LIN {X 0,Y 249.727,Z 1176.579,A -85,B 0,C 180,E1 12706.065,E2 12706.065} C_VEL
LIN {X 0,Y 248.616,Z 1179.166,A -85,B 0,C 180,E1 12701.365,E2 12701.365} C_VEL
LIN {X 0,Y 248.168,Z 1180.788,A -85,B 0,C 180,E1 12696.942,E2 12696.942} C_VEL
LIN {X 0,Y 248.027,Z 1181.611,A -85,B 0,C 180,E1 12692.773,E2 12692.773} C_VEL
LIN {X 0,Y 248.02,Z 1181.751,A -85,B 0,C 180,E1 12688.614,E2 12688.614} C_VEL
LIN {X 0,Y 248.114,Z 1181.08,A -85,B 0,C 180,E1 12683.986,E2 12683.986} C_VEL
LIN {X 0,Y 248.534,Z 1179.438,A -85,B 0,C 180,E1 12679.101,E2 12679.101} C_VEL
LIN {X 0,Y 249.624,Z 1176.826,A -85,B 0,C 180,E1 12674.195,E2 12674.195} C_VEL
LIN {X 0,Y 251.654,Z 1173.217,A -85,B 0,C 180,E1 12669.292,E2 12669.292} C_VEL
LIN {X 0,Y 254.855,Z 1168.577,A -85,B 0,C 180,E1 12664.434,E2 12664.434} C_VEL
LIN {X 0,Y 259.34,Z 1162.869,A -85,B 0,C 180,E1 12659.665,E2 12659.665} C_VEL
LIN {X 0,Y 266.478,Z 1154.638,A -85,B 0,C 180,E1 12654.144,E2 12654.144} C_VEL
LIN {X 0,Y 275.857,Z 1144.197,A -85,B 0,C 180,E1 12648.726,E2 12648.726} C_VEL
LIN {X 0,Y 284.944,Z 1134.318,A -85,B 0,C 180,E1 12644.573,E2 12644.573} C_VEL
LIN {X 0,Y 294.763,Z 1123.639,A -85,B 0,C 180,E1 12640.849,E2 12640.849} C_VEL
LIN {X 0,Y 307.374,Z 1109.73,A -85,B 0,C 180,E1 12636.85,E2 12636.85} C_VEL
LIN {X 0,Y 320.654,Z 1094.237,A -85,B 0,C 180,E1 12633.286,E2 12633.286} C_VEL
LIN {X 0,Y 332.217,Z 1080.145,A -85,B 0,C 180,E1 12630.598,E2 12630.598} C_VEL
LIN {X 0,Y 343.091,Z 1066.216,A -85,B 0,C 180,E1 12628.345,E2 12628.345} C_VEL
LIN {X 0,Y 354.794,Z 1050.336,A -85,B 0,C 180,E1 12626.159,E2 12626.159} C_VEL
LIN {X 0,Y 368.74,Z 1030.057,A -85,B 0,C 180,E1 12623.831,E2 12623.831} C_VEL
LIN {X 0,Y 381.488,Z 1009.491,A -85,B 0,C 180,E1 12621.904,E2 12621.904} C_VEL
LIN {X 0,Y 391.938,Z 991.177,A -85,B 0,C 180,E1 12620.457,E2 12620.457} C_VEL
LIN {X 0,Y 401.368,Z 973.16,A -85,B 0,C 180,E1 12619.242,E2 12619.242} C_VEL
LIN {X 0,Y 411.167,Z 952.497,A -85,B 0,C 180,E1 12618.045,E2 12618.045} C_VEL
LIN {X 0,Y 422.058,Z 926.302,A -85,B 0,C 180,E1 12616.8,E2 12616.8} C_VEL
LIN {X 0,Y 429.551,Z 905.47,A -85,B 0,C 180,E1 12615.986,E2 12615.986} C_VEL
LIN {X 0,Y 435.925,Z 885.156,A -85,B 0,C 180,E1 12615.318,E2 12615.318} C_VEL
LIN {X 0,Y 441.618,Z 863.935,A -85,B 0,C 180,E1 12614.735,E2 12614.735} C_VEL
LIN {X 0,Y 445.99,Z 844.495,A -85,B 0,C 180,E1 12614.298,E2 12614.298} C_VEL
LIN {X 0,Y 447.312,Z 837.117,A -85,B 0,C 180,E1 12614.033,E2 12614.033} C_VEL
LIN {X 0,Y 449.125,Z 817.839,A -85,B 0,C 180,E1 12612.916,E2 12612.916} C_VEL
LIN {X 0,Y 449.804,Z 811.396,A -85,B 0,C 180,E1 12612.724,E2 12612.724} C_VEL
LIN {X 0,Y 456.299,Z 750.449,A -85,B 0,C 180,E1 12611.84,E2 12611.84} C_VEL
LIN {X 0,Y 471.03,Z 607.918,A -85,B 0,C 180,E1 12609.811,E2 12609.811} C_VEL
LIN {X 0,Y 468.952,Z 603.858,A -85,B 0,C 180,E1 12607.72,E2 12607.72} C_VEL
LIN {X 0,Y 467.352,Z 600.49,A -85,B 0,C 180,E1 12605.525,E2 12605.525} C_VEL
LIN {X 0,Y 465.914,Z 596.286,A -85,B 0,C 180,E1 12601.107,E2 12601.107} C_VEL
LIN {X 0,Y 465.917,Z 596.314,A -85,B 0,C 180,E1 12599.262,E2 12599.262} C_VEL
LIN {X 0,Y 467.226,Z 600.314,A -85,B 0,C 180,E1 12595.089,E2 12595.089} C_VEL
LIN {X 0,Y 467.857,Z 601.547,A -85,B 0,C 180,E1 12594.112,E2 12594.112} C_VEL
LIN {X 0,Y 470.021,Z 605.91,A -85,B 0,C 180,E1 12591.559,E2 12591.559} C_VEL
LIN {X 0,Y 471.151,Z 608.251,A -85,B 0,C 180,E1 12590.489,E2 12590.489} C_VEL
LIN {X 0,Y 449.874,Z 813.61,A -85,B 0,C 180,E1 12587.551,E2 12587.551} C_VEL
LIN {X 0,Y 446.454,Z 836.613,A -85,B 0,C 180,E1 12587.182,E2 12587.182} C_VEL
LIN {X 0,Y 440.618,Z 864.958,A -85,B 0,C 180,E1 12586.666,E2 12586.666} C_VEL
LIN {X 0,Y 434.14,Z 889.147,A -85,B 0,C 180,E1 12586.106,E2 12586.106} C_VEL
LIN {X 0,Y 427.55,Z 910.072,A -85,B 0,C 180,E1 12585.504,E2 12585.504} C_VEL
LIN {X 0,Y 420.15,Z 930.562,A -85,B 0,C 180,E1 12584.794,E2 12584.794} C_VEL
LIN {X 0,Y 411.591,Z 951.546,A -85,B 0,C 180,E1 12583.922,E2 12583.922} C_VEL
LIN {X 0,Y 399.271,Z 978.022,A -85,B 0,C 180,E1 12582.573,E2 12582.573} C_VEL
LIN {X 0,Y 388.486,Z 998.548,A -85,B 0,C 180,E1 12581.286,E2 12581.286} C_VEL
LIN {X 0,Y 378.298,Z 1016.269,A -85,B 0,C 180,E1 12579.984,E2 12579.984} C_VEL
LIN {X 0,Y 367.137,Z 1034.234,A -85,B 0,C 180,E1 12578.428,E2 12578.428} C_VEL
LIN {X 0,Y 353.455,Z 1054.661,A -85,B 0,C 180,E1 12576.315,E2 12576.315} C_VEL
LIN {X 0,Y 338.832,Z 1074.514,A -85,B 0,C 180,E1 12573.776,E2 12573.776} C_VEL
LIN {X 0,Y 326.822,Z 1089.878,A -85,B 0,C 180,E1 12571.405,E2 12571.405} C_VEL
LIN {X 0,Y 315.399,Z 1103.791,A -85,B 0,C 180,E1 12568.863,E2 12568.863} C_VEL
LIN {X 0,Y 303.391,Z 1117.825,A -85,B 0,C 180,E1 12565.812,E2 12565.812} C_VEL
LIN {X 0,Y 288.384,Z 1134.661,A -85,B 0,C 180,E1 12561.269,E2 12561.269} C_VEL
LIN {X 0,Y 277.619,Z 1146.477,A -85,B 0,C 180,E1 12557.283,E2 12557.283} C_VEL
LIN {X 0,Y 268.578,Z 1156.436,A -85,B 0,C 180,E1 12553.235,E2 12553.235} C_VEL
LIN {X 0,Y 260.061,Z 1166.03,A -85,B 0,C 180,E1 12548.524,E2 12548.524} C_VEL
LIN {X 0,Y 251.434,Z 1176.35,A -85,B 0,C 180,E1 12542.107,E2 12542.107} C_VEL
LIN {X 0,Y 246.423,Z 1183.046,A -85,B 0,C 180,E1 12536.768,E2 12536.768} C_VEL
LIN {X 0,Y 243.201,Z 1188.116,A -85,B 0,C 180,E1 12531.716,E2 12531.716} C_VEL
LIN {X 0,Y 241.293,Z 1191.973,A -85,B 0,C 180,E1 12526.815,E2 12526.815} C_VEL
LIN {X 0,Y 240.319,Z 1194.802,A -85,B 0,C 180,E1 12522.007,E2 12522.007} C_VEL
LIN {X 0,Y 240.037,Z 1196.639,A -85,B 0,C 180,E1 12517.419,E2 12517.419} C_VEL
LIN {X 0,Y 240.009,Z 1197.592,A -85,B 0,C 180,E1 12513.104,E2 12513.104} C_VEL
LIN {X 0,Y 240.02,Z 1197.782,A -85,B 0,C 180,E1 12508.807,E2 12508.807} C_VEL
LIN {X 0,Y 240.006,Z 1197.061,A -85,B 0,C 180,E1 12504.022,E2 12504.022} C_VEL
LIN {X 0,Y 240.223,Z 1195.267,A -85,B 0,C 180,E1 12498.962,E2 12498.962} C_VEL
LIN {X 0,Y 241.106,Z 1192.425,A -85,B 0,C 180,E1 12493.868,E2 12493.868} C_VEL
LIN {X 0,Y 242.957,Z 1188.524,A -85,B 0,C 180,E1 12488.768,E2 12488.768} C_VEL
LIN {X 0,Y 246.061,Z 1183.545,A -85,B 0,C 180,E1 12483.71,E2 12483.71} C_VEL
LIN {X 0,Y 250.51,Z 1177.46,A -85,B 0,C 180,E1 12478.744,E2 12478.744} C_VEL
LIN {X 0,Y 257.044,Z 1169.504,A -85,B 0,C 180,E1 12473.477,E2 12473.477} C_VEL
LIN {X 0,Y 267.323,Z 1157.79,A -85,B 0,C 180,E1 12467.392,E2 12467.392} C_VEL
LIN {X 0,Y 276.776,Z 1147.339,A -85,B 0,C 180,E1 12463.062,E2 12463.062} C_VEL
LIN {X 0,Y 286.761,Z 1136.342,A -85,B 0,C 180,E1 12459.281,E2 12459.281} C_VEL
LIN {X 0,Y 299.166,Z 1122.555,A -85,B 0,C 180,E1 12455.365,E2 12455.365} C_VEL
LIN {X 0,Y 313.835,Z 1105.53,A -85,B 0,C 180,E1 12451.501,E2 12451.501} C_VEL
LIN {X 0,Y 326.118,Z 1090.599,A -85,B 0,C 180,E1 12448.735,E2 12448.735} C_VEL
LIN {X 0,Y 338.094,Z 1075.298,A -85,B 0,C 180,E1 12446.354,E2 12446.354} C_VEL
LIN {X 0,Y 352.128,Z 1056.313,A -85,B 0,C 180,E1 12443.892,E2 12443.892} C_VEL
LIN {X 0,Y 366.36,Z 1035.204,A -85,B 0,C 180,E1 12441.677,E2 12441.677} C_VEL
LIN {X 0,Y 377.88,Z 1016.689,A -85,B 0,C 180,E1 12440.063,E2 12440.063} C_VEL
LIN {X 0,Y 388.469,Z 998.262,A -85,B 0,C 180,E1 12438.707,E2 12438.707} C_VEL
LIN {X 0,Y 399.677,Z 976.889,A -85,B 0,C 180,E1 12437.373,E2 12437.373} C_VEL
LIN {X 0,Y 411.443,Z 951.467,A -85,B 0,C 180,E1 12436.084,E2 12436.084} C_VEL
LIN {X 0,Y 420.134,Z 930.114,A -85,B 0,C 180,E1 12435.197,E2 12435.197} C_VEL
LIN {X 0,Y 427.534,Z 909.552,A -85,B 0,C 180,E1 12434.487,E2 12434.487} C_VEL
LIN {X 0,Y 434.347,Z 887.8,A -85,B 0,C 180,E1 12433.867,E2 12433.867} C_VEL
LIN {X 0,Y 441.555,Z 860.083,A -85,B 0,C 180,E1 12433.243,E2 12433.243} C_VEL
LIN {X 0,Y 446.555,Z 834.801,A -85,B 0,C 180,E1 12432.794,E2 12432.794} C_VEL
LIN {X 0,Y 449.81,Z 812.463,A -85,B 0,C 180,E1 12432.437,E2 12432.437} C_VEL
LIN {X 0,Y 470.962,Z 607.908,A -85,B 0,C 180,E1 12429.509,E2 12429.509} C_VEL
LIN {X 0,Y 468.889,Z 603.932,A -85,B 0,C 180,E1 12427.474,E2 12427.474} C_VEL
LIN {X 0,Y 467.155,Z 600.324,A -85,B 0,C 180,E1 12425.158,E2 12425.158} C_VEL
LIN {X 0,Y 465.714,Z 596.603,A -85,B 0,C 180,E1 12421.353,E2 12421.353} C_VEL
LIN {X 0,Y 465.647,Z 596.093,A -85,B 0,C 180,E1 12420.615,E2 12420.615} C_VEL
LIN {X 0,Y 465.682,Z 596.236,A -85,B 0,C 180,E1 12418.524,E2 12418.524} C_VEL
LIN {X 0,Y 467.54,Z 601.157,A -85,B 0,C 180,E1 12413.738,E2 12413.738} C_VEL
LIN {X 0,Y 469.614,Z 605.388,A -85,B 0,C 180,E1 12411.243,E2 12411.243} C_VEL
LIN {X 0,Y 470.81,Z 607.98,A -85,B 0,C 180,E1 12410.086,E2 12410.086} C_VEL
LIN {X 0,Y 449.965,Z 808.417,A -85,B 0,C 180,E1 12407.225,E2 12407.225} C_VEL
LIN {X 0,Y 446.124,Z 833.492,A -85,B 0,C 180,E1 12406.821,E2 12406.821} C_VEL
LIN {X 0,Y 440.07,Z 861.713,A -85,B 0,C 180,E1 12406.239,E2 12406.239} C_VEL
LIN {X 0,Y 434.212,Z 883.569,A -85,B 0,C 180,E1 12405.663,E2 12405.663} C_VEL
LIN {X 0,Y 427.959,Z 903.481,A -85,B 0,C 180,E1 12405.033,E2 12405.033} C_VEL
LIN {X 0,Y 420.689,Z 923.691,A -85,B 0,C 180,E1 12404.273,E2 12404.273} C_VEL
LIN {X 0,Y 411.386,Z 946.458,A -85,B 0,C 180,E1 12403.256,E2 12403.256} C_VEL
LIN {X 0,Y 399.73,Z 971.175,A -85,B 0,C 180,E1 12401.898,E2 12401.898} C_VEL
LIN {X 0,Y 389.529,Z 990.45,A -85,B 0,C 180,E1 12400.637,E2 12400.637} C_VEL
LIN {X 0,Y 379.06,Z 1008.555,A -85,B 0,C 180,E1 12399.24,E2 12399.24} C_VEL
LIN {X 0,Y 367.699,Z 1026.642,A -85,B 0,C 180,E1 12397.598,E2 12397.598} C_VEL
LIN {X 0,Y 352.89,Z 1048.188,A -85,B 0,C 180,E1 12395.242,E2 12395.242} C_VEL
LIN {X 0,Y 340.117,Z 1065.189,A -85,B 0,C 180,E1 12392.966,E2 12392.966} C_VEL
LIN {X 0,Y 328.91,Z 1079.228,A -85,B 0,C 180,E1 12390.745,E2 12390.745} C_VEL
LIN {X 0,Y 317.549,Z 1092.731,A -85,B 0,C 180,E1 12388.227,E2 12388.227} C_VEL
LIN {X 0,Y 305.594,Z 1106.31,A -85,B 0,C 180,E1 12385.208,E2 12385.208} C_VEL
LIN {X 0,Y 291.164,Z 1121.982,A -85,B 0,C 180,E1 12380.903,E2 12380.903} C_VEL
LIN {X 0,Y 280.268,Z 1133.369,A -85,B 0,C 180,E1 12376.999,E2 12376.999} C_VEL
LIN {X 0,Y 271.036,Z 1142.926,A -85,B 0,C 180,E1 12373.037,E2 12373.037} C_VEL
LIN {X 0,Y 262.669,Z 1151.691,A -85,B 0,C 180,E1 12368.629,E2 12368.629} C_VEL
LIN {X 0,Y 254.223,Z 1160.944,A -85,B 0,C 180,E1 12362.871,E2 12362.871} C_VEL
LIN {X 0,Y 247.901,Z 1168.239,A -85,B 0,C 180,E1 12356.855,E2 12356.855} C_VEL
LIN {X 0,Y 244.17,Z 1173.191,A -85,B 0,C 180,E1 12351.626,E2 12351.626} C_VEL
LIN {X 0,Y 241.887,Z 1176.865,A -85,B 0,C 180,E1 12346.572,E2 12346.572} C_VEL
LIN {X 0,Y 240.683,Z 1179.432,A -85,B 0,C 180,E1 12341.745,E2 12341.745} C_VEL
LIN {X 0,Y 240.186,Z 1181.052,A -85,B 0,C 180,E1 12337.174,E2 12337.174} C_VEL
LIN {X 0,Y 240.033,Z 1181.874,A -85,B 0,C 180,E1 12332.865,E2 12332.865} C_VEL
LIN {X 0,Y 240.025,Z 1182.013,A -85,B 0,C 180,E1 12328.568,E2 12328.568} C_VEL
LIN {X 0,Y 240.129,Z 1181.343,A -85,B 0,C 180,E1 12323.785,E2 12323.785} C_VEL
LIN {X 0,Y 240.592,Z 1179.703,A -85,B 0,C 180,E1 12318.736,E2 12318.736} C_VEL
LIN {X 0,Y 241.801,Z 1177.057,A -85,B 0,C 180,E1 12313.611,E2 12313.611} C_VEL
LIN {X 0,Y 243.989,Z 1173.486,A -85,B 0,C 180,E1 12308.61,E2 12308.61} C_VEL
LIN {X 0,Y 247.426,Z 1168.847,A -85,B 0,C 180,E1 12303.608,E2 12303.608} C_VEL
LIN {X 0,Y 252.207,Z 1163.141,A -85,B 0,C 180,E1 12298.712,E2 12298.712} C_VEL
LIN {X 0,Y 259.734,Z 1154.949,A -85,B 0,C 180,E1 12293.092,E2 12293.092} C_VEL
LIN {X 0,Y 269.634,Z 1144.47,A -85,B 0,C 180,E1 12287.554,E2 12287.554} C_VEL
LIN {X 0,Y 279.146,Z 1134.596,A -85,B 0,C 180,E1 12283.355,E2 12283.355} C_VEL
LIN {X 0,Y 289.38,Z 1123.911,A -85,B 0,C 180,E1 12279.601,E2 12279.601} C_VEL
LIN {X 0,Y 302.487,Z 1109.963,A -85,B 0,C 180,E1 12275.576,E2 12275.576} C_VEL
LIN {X 0,Y 316.108,Z 1094.573,A -85,B 0,C 180,E1 12272.039,E2 12272.039} C_VEL
LIN {X 0,Y 328.073,Z 1080.415,A -85,B 0,C 180,E1 12269.351,E2 12269.351} C_VEL
LIN {X 0,Y 339.246,Z 1066.484,A -85,B 0,C 180,E1 12267.117,E2 12267.117} C_VEL
LIN {X 0,Y 350.868,Z 1051.103,A -85,B 0,C 180,E1 12265.016,E2 12265.016} C_VEL
LIN {X 0,Y 365.112,Z 1030.929,A -85,B 0,C 180,E1 12262.715,E2 12262.715} C_VEL
LIN {X 0,Y 378.514,Z 1009.755,A -85,B 0,C 180,E1 12260.756,E2 12260.756} C_VEL
LIN {X 0,Y 388.941,Z 991.838,A -85,B 0,C 180,E1 12259.361,E2 12259.361} C_VEL
LIN {X 0,Y 398.351,Z 974.227,A -85,B 0,C 180,E1 12258.19,E2 12258.19} C_VEL
LIN {X 0,Y 407.47,Z 955.44,A -85,B 0,C 180,E1 12257.107,E2 12257.107} C_VEL
LIN {X 0,Y 418.014,Z 931.249,A -85,B 0,C 180,E1 12255.94,E2 12255.94} C_VEL
LIN {X 0,Y 426.974,Z 907.004,A -85,B 0,C 180,E1 12254.992,E2 12254.992} C_VEL
LIN {X 0,Y 433.654,Z 886.148,A -85,B 0,C 180,E1 12254.315,E2 12254.315} C_VEL
LIN {X 0,Y 439.482,Z 864.836,A -85,B 0,C 180,E1 12253.739,E2 12253.739} C_VEL
LIN {X 0,Y 444.549,Z 842.515,A -85,B 0,C 180,E1 12253.252,E2 12253.252} C_VEL
LIN {X 0,Y 449.48,Z 814.028,A -85,B 0,C 180,E1 12252.763,E2 12252.763} C_VEL
LIN {X 0,Y 449.804,Z 811.396,A -85,B 0,C 180,E1 12252.724,E2 12252.724} C_VEL
LIN {X 0,Y 450.526,Z 803.885,A -85,B 0,C 180,E1 12252.49,E2 12252.49} C_VEL
LIN {X 0,Y 451.401,Z 784.372,A -85,B 0,C 180,E1 12251.427,E2 12251.427} C_VEL
LIN {X 0,Y 451.905,Z 777.899,A -85,B 0,C 180,E1 12251.237,E2 12251.237} C_VEL
LIN {X 0,Y 469.061,Z 614.281,A -85,B 0,C 180,E1 12248.921,E2 12248.921} C_VEL
LIN {X 0,Y 467.756,Z 611.57,A -85,B 0,C 180,E1 12247.492,E2 12247.492} C_VEL
LIN {X 0,Y 466.218,Z 608.279,A -85,B 0,C 180,E1 12245.291,E2 12245.291} C_VEL
LIN {X 0,Y 464.923,Z 604.057,A -85,B 0,C 180,E1 12240.739,E2 12240.739} C_VEL
LIN {X 0,Y 464.933,Z 604.329,A -85,B 0,C 180,E1 12239.261,E2 12239.261} C_VEL
LIN {X 0,Y 466.251,Z 608.287,A -85,B 0,C 180,E1 12235.079,E2 12235.079} C_VEL
LIN {X 0,Y 466.989,Z 609.985,A -85,B 0,C 180,E1 12233.916,E2 12233.916} C_VEL
LIN {X 0,Y 468.79,Z 613.597,A -85,B 0,C 180,E1 12231.784,E2 12231.784} C_VEL
LIN {X 0,Y 469.179,Z 614.647,A -85,B 0,C 180,E1 12231.366,E2 12231.366} C_VEL
LIN {X 0,Y 448.075,Z 814.43,A -85,B 0,C 180,E1 12228.541,E2 12228.541} C_VEL
LIN {X 0,Y 444.253,Z 839.22,A -85,B 0,C 180,E1 12228.147,E2 12228.147} C_VEL
LIN {X 0,Y 437.953,Z 868.083,A -85,B 0,C 180,E1 12227.62,E2 12227.62} C_VEL
LIN {X 0,Y 432.048,Z 889.633,A -85,B 0,C 180,E1 12227.127,E2 12227.127} C_VEL
LIN {X 0,Y 425.417,Z 910.328,A -85,B 0,C 180,E1 12226.545,E2 12226.545} C_VEL
LIN {X 0,Y 417.653,Z 931.439,A -85,B 0,C 180,E1 12225.827,E2 12225.827} C_VEL
LIN {X 0,Y 407.204,Z 956.413,A -85,B 0,C 180,E1 12224.792,E2 12224.792} C_VEL
LIN {X 0,Y 396.041,Z 979.393,A -85,B 0,C 180,E1 12223.609,E2 12223.609} C_VEL
LIN {X 0,Y 385.924,Z 998.282,A -85,B 0,C 180,E1 12222.443,E2 12222.443} C_VEL
LIN {X 0,Y 375.549,Z 1016.001,A -85,B 0,C 180,E1 12221.169,E2 12221.169} C_VEL
LIN {X 0,Y 364.195,Z 1033.929,A -85,B 0,C 180,E1 12219.644,E2 12219.644} C_VEL
LIN {X 0,Y 350.017,Z 1054.65,A -85,B 0,C 180,E1 12217.534,E2 12217.534} C_VEL
LIN {X 0,Y 335.031,Z 1074.483,A -85,B 0,C 180,E1 12215.024,E2 12215.024} C_VEL
LIN {X 0,Y 322.893,Z 1089.606,A -85,B 0,C 180,E1 12212.712,E2 12212.712} C_VEL
LIN {X 0,Y 311.131,Z 1103.517,A -85,B 0,C 180,E1 12210.19,E2 12210.19} C_VEL
LIN {X 0,Y 298.734,Z 1117.551,A -85,B 0,C 180,E1 12207.15,E2 12207.15} C_VEL
LIN {X 0,Y 283.173,Z 1134.387,A -85,B 0,C 180,E1 12202.603,E2 12202.603} C_VEL
LIN {X 0,Y 271.947,Z 1146.201,A -85,B 0,C 180,E1 12198.594,E2 12198.594} C_VEL
LIN {X 0,Y 262.475,Z 1156.159,A -85,B 0,C 180,E1 12194.501,E2 12194.501} C_VEL
LIN {X 0,Y 253.522,Z 1165.755,A -85,B 0,C 180,E1 12189.71,E2 12189.71} C_VEL
LIN {X 0,Y 244.46,Z 1175.968,A -85,B 0,C 180,E1 12183.235,E2 12183.235} C_VEL
LIN {X 0,Y 238.998,Z 1182.773,A -85,B 0,C 180,E1 12177.669,E2 12177.669} C_VEL
LIN {X 0,Y 235.533,Z 1187.845,A -85,B 0,C 180,E1 12172.461,E2 12172.461} C_VEL
LIN {X 0,Y 233.459,Z 1191.672,A -85,B 0,C 180,E1 12167.445,E2 12167.445} C_VEL
LIN {X 0,Y 232.402,Z 1194.415,A -85,B 0,C 180,E1 12162.675,E2 12162.675} C_VEL
LIN {X 0,Y 232.049,Z 1196.302,A -85,B 0,C 180,E1 12157.925,E2 12157.925} C_VEL
LIN {X 0,Y 232.009,Z 1197.305,A -85,B 0,C 180,E1 12153.459,E2 12153.459} C_VEL
LIN {X 0,Y 232.024,Z 1197.519,A -85,B 0,C 180,E1 12148.765,E2 12148.765} C_VEL
LIN {X 0,Y 232.011,Z 1196.797,A -85,B 0,C 180,E1 12143.815,E2 12143.815} C_VEL
LIN {X 0,Y 232.257,Z 1195,A -85,B 0,C 180,E1 12138.578,E2 12138.578} C_VEL
LIN {X 0,Y 233.239,Z 1192.155,A -85,B 0,C 180,E1 12133.309,E2 12133.309} C_VEL
LIN {X 0,Y 235.269,Z 1188.252,A -85,B 0,C 180,E1 12128.038,E2 12128.038} C_VEL
LIN {X 0,Y 238.612,Z 1183.271,A -85,B 0,C 180,E1 12122.823,E2 12122.823} C_VEL
LIN {X 0,Y 243.381,Z 1177.183,A -85,B 0,C 180,E1 12117.719,E2 12117.719} C_VEL
LIN {X 0,Y 250.321,Z 1169.226,A -85,B 0,C 180,E1 12112.329,E2 12112.329} C_VEL
LIN {X 0,Y 261.167,Z 1157.512,A -85,B 0,C 180,E1 12106.137,E2 12106.137} C_VEL
LIN {X 0,Y 270.942,Z 1147.188,A -85,B 0,C 180,E1 12101.803,E2 12101.803} C_VEL
LIN {X 0,Y 280.926,Z 1136.648,A -85,B 0,C 180,E1 12098.134,E2 12098.134} C_VEL
LIN {X 0,Y 292.525,Z 1124.219,A -85,B 0,C 180,E1 12094.539,E2 12094.539} C_VEL
LIN {X 0,Y 307.773,Z 1107.307,A -85,B 0,C 180,E1 12090.582,E2 12090.582} C_VEL
LIN {X 0,Y 321.462,Z 1091.179,A -85,B 0,C 180,E1 12087.57,E2 12087.57} C_VEL
LIN {X 0,Y 333.725,Z 1075.96,A -85,B 0,C 180,E1 12085.203,E2 12085.203} C_VEL
LIN {X 0,Y 346.134,Z 1059.629,A -85,B 0,C 180,E1 12083.07,E2 12083.07} C_VEL
LIN {X 0,Y 361.386,Z 1038.003,A -85,B 0,C 180,E1 12080.747,E2 12080.747} C_VEL
LIN {X 0,Y 374.306,Z 1017.762,A -85,B 0,C 180,E1 12078.983,E2 12078.983} C_VEL
LIN {X 0,Y 385.072,Z 999.469,A -85,B 0,C 180,E1 12077.649,E2 12077.649} C_VEL
LIN {X 0,Y 395.391,Z 980.285,A -85,B 0,C 180,E1 12076.453,E2 12076.453} C_VEL
LIN {X 0,Y 407.188,Z 956.034,A -85,B 0,C 180,E1 12075.2,E2 12075.2} C_VEL
LIN {X 0,Y 417.2,Z 932.115,A -85,B 0,C 180,E1 12074.207,E2 12074.207} C_VEL
LIN {X 0,Y 424.968,Z 911.058,A -85,B 0,C 180,E1 12073.486,E2 12073.486} C_VEL
LIN {X 0,Y 431.81,Z 889.754,A -85,B 0,C 180,E1 12072.884,E2 12072.884} C_VEL
LIN {X 0,Y 438.091,Z 866.761,A -85,B 0,C 180,E1 12072.36,E2 12072.36} C_VEL
LIN {X 0,Y 444.399,Z 837.128,A -85,B 0,C 180,E1 12071.825,E2 12071.825} C_VEL
LIN {X 0,Y 447.945,Z 813.767,A -85,B 0,C 180,E1 12071.455,E2 12071.455} C_VEL
LIN {X 0,Y 468.989,Z 614.287,A -85,B 0,C 180,E1 12068.633,E2 12068.633} C_VEL
LIN {X 0,Y 467.578,Z 611.457,A -85,B 0,C 180,E1 12067.125,E2 12067.125} C_VEL
LIN {X 0,Y 466.098,Z 608.204,A -85,B 0,C 180,E1 12065.046,E2 12065.046} C_VEL
LIN {X 0,Y 464.719,Z 604.483,A -85,B 0,C 180,E1 12061.233,E2 12061.233} C_VEL
LIN {X 0,Y 464.657,Z 604.037,A -85,B 0,C 180,E1 12060.493,E2 12060.493} C_VEL
LIN {X 0,Y 464.696,Z 604.266,A -85,B 0,C 180,E1 12058.52,E2 12058.52} C_VEL
LIN {X 0,Y 466.432,Z 608.961,A -85,B 0,C 180,E1 12053.909,E2 12053.909} C_VEL
LIN {X 0,Y 468.445,Z 613.211,A -85,B 0,C 180,E1 12051.407,E2 12051.407} C_VEL
LIN {X 0,Y 468.847,Z 614.358,A -85,B 0,C 180,E1 12050.964,E2 12050.964} C_VEL
LIN {X 0,Y 448.25,Z 808.808,A -85,B 0,C 180,E1 12048.221,E2 12048.221} C_VEL
LIN {X 0,Y 444.285,Z 834.257,A -85,B 0,C 180,E1 12047.818,E2 12047.818} C_VEL
LIN {X 0,Y 438.204,Z 862.095,A -85,B 0,C 180,E1 12047.255,E2 12047.255} C_VEL
LIN {X 0,Y 432.292,Z 883.842,A -85,B 0,C 180,E1 12046.695,E2 12046.695} C_VEL
LIN {X 0,Y 425.95,Z 903.753,A -85,B 0,C 180,E1 12046.079,E2 12046.079} C_VEL
LIN {X 0,Y 418.51,Z 924.131,A -85,B 0,C 180,E1 12045.33,E2 12045.33} C_VEL
LIN {X 0,Y 408.703,Z 947.728,A -85,B 0,C 180,E1 12044.294,E2 12044.294} C_VEL
LIN {X 0,Y 397.28,Z 971.447,A -85,B 0,C 180,E1 12043.012,E2 12043.012} C_VEL
LIN {X 0,Y 386.929,Z 990.678,A -85,B 0,C 180,E1 12041.779,E2 12041.779} C_VEL
LIN {X 0,Y 376.242,Z 1008.827,A -85,B 0,C 180,E1 12040.403,E2 12040.403} C_VEL
LIN {X 0,Y 365.182,Z 1026.11,A -85,B 0,C 180,E1 12038.866,E2 12038.866} C_VEL
LIN {X 0,Y 351.017,Z 1046.51,A -85,B 0,C 180,E1 12036.705,E2 12036.705} C_VEL
LIN {X 0,Y 337.089,Z 1064.659,A -85,B 0,C 180,E1 12034.337,E2 12034.337} C_VEL
LIN {X 0,Y 324.938,Z 1079.503,A -85,B 0,C 180,E1 12032.021,E2 12032.021} C_VEL
LIN {X 0,Y 313.1,Z 1093.179,A -85,B 0,C 180,E1 12029.484,E2 12029.484} C_VEL
LIN {X 0,Y 300.296,Z 1107.273,A -85,B 0,C 180,E1 12026.345,E2 12026.345} C_VEL
LIN {X 0,Y 285.411,Z 1122.819,A -85,B 0,C 180,E1 12022.02,E2 12022.02} C_VEL
LIN {X 0,Y 274.137,Z 1134.147,A -85,B 0,C 180,E1 12018.077,E2 12018.077} C_VEL
LIN {X 0,Y 264.55,Z 1143.649,A -85,B 0,C 180,E1 12014.061,E2 12014.061} C_VEL
LIN {X 0,Y 255.822,Z 1152.36,A -85,B 0,C 180,E1 12009.574,E2 12009.574} C_VEL
LIN {X 0,Y 246.532,Z 1161.958,A -85,B 0,C 180,E1 12003.332,E2 12003.332} C_VEL
LIN {X 0,Y 240.339,Z 1168.756,A -85,B 0,C 180,E1 11997.502,E2 11997.502} C_VEL
LIN {X 0,Y 236.546,Z 1173.462,A -85,B 0,C 180,E1 11992.36,E2 11992.36} C_VEL
LIN {X 0,Y 234.074,Z 1177.134,A -85,B 0,C 180,E1 11987.142,E2 11987.142} C_VEL
LIN {X 0,Y 232.754,Z 1179.699,A -85,B 0,C 180,E1 11982.151,E2 11982.151} C_VEL
LIN {X 0,Y 232.206,Z 1181.316,A -85,B 0,C 180,E1 11977.422,E2 11977.422} C_VEL
LIN {X 0,Y 232.039,Z 1182.136,A -85,B 0,C 180,E1 11972.964,E2 11972.964} C_VEL
LIN {X 0,Y 232.029,Z 1182.276,A -85,B 0,C 180,E1 11968.518,E2 11968.518} C_VEL
LIN {X 0,Y 232.145,Z 1181.607,A -85,B 0,C 180,E1 11963.57,E2 11963.57} C_VEL
LIN {X 0,Y 232.657,Z 1179.969,A -85,B 0,C 180,E1 11958.347,E2 11958.347} C_VEL
LIN {X 0,Y 233.958,Z 1177.361,A -85,B 0,C 180,E1 11953.106,E2 11953.106} C_VEL
LIN {X 0,Y 236.355,Z 1173.755,A -85,B 0,C 180,E1 11947.883,E2 11947.883} C_VEL
LIN {X 0,Y 240.056,Z 1169.117,A -85,B 0,C 180,E1 11942.732,E2 11942.732} C_VEL
LIN {X 0,Y 245.43,Z 1163.119,A -85,B 0,C 180,E1 11937.469,E2 11937.469} C_VEL
LIN {X 0,Y 253.856,Z 1154.513,A -85,B 0,C 180,E1 11931.515,E2 11931.515} C_VEL
LIN {X 0,Y 263.977,Z 1144.295,A -85,B 0,C 180,E1 11926.121,E2 11926.121} C_VEL
LIN {X 0,Y 273.489,Z 1134.868,A -85,B 0,C 180,E1 11922.085,E2 11922.085} C_VEL
LIN {X 0,Y 283.578,Z 1124.744,A -85,B 0,C 180,E1 11918.488,E2 11918.488} C_VEL
LIN {X 0,Y 295.491,Z 1112.49,A -85,B 0,C 180,E1 11914.881,E2 11914.881} C_VEL
LIN {X 0,Y 311.114,Z 1095.601,A -85,B 0,C 180,E1 11910.898,E2 11910.898} C_VEL
LIN {X 0,Y 323.389,Z 1081.517,A -85,B 0,C 180,E1 11908.217,E2 11908.217} C_VEL
LIN {X 0,Y 335.56,Z 1066.753,A -85,B 0,C 180,E1 11905.861,E2 11905.861} C_VEL
LIN {X 0,Y 347.466,Z 1051.37,A -85,B 0,C 180,E1 11903.785,E2 11903.785} C_VEL
LIN {X 0,Y 361.605,Z 1031.79,A -85,B 0,C 180,E1 11901.578,E2 11901.578} C_VEL
LIN {X 0,Y 375.331,Z 1010.614,A -85,B 0,C 180,E1 11899.639,E2 11899.639} C_VEL
LIN {X 0,Y 386.313,Z 992.101,A -85,B 0,C 180,E1 11898.219,E2 11898.219} C_VEL
LIN {X 0,Y 396.308,Z 973.683,A -85,B 0,C 180,E1 11897.023,E2 11897.023} C_VEL
LIN {X 0,Y 406.438,Z 953.018,A -85,B 0,C 180,E1 11895.872,E2 11895.872} C_VEL
LIN {X 0,Y 417.588,Z 927.05,A -85,B 0,C 180,E1 11894.688,E2 11894.688} C_VEL
LIN {X 0,Y 425.395,Z 905.983,A -85,B 0,C 180,E1 11893.899,E2 11893.899} C_VEL
LIN {X 0,Y 432.141,Z 885.042,A -85,B 0,C 180,E1 11893.242,E2 11893.242} C_VEL
LIN {X 0,Y 438.005,Z 863.682,A -85,B 0,C 180,E1 11892.686,E2 11892.686} C_VEL
LIN {X 0,Y 443.734,Z 838.321,A -85,B 0,C 180,E1 11892.158,E2 11892.158} C_VEL
LIN {X 0,Y 448.274,Z 810.317,A -85,B 0,C 180,E1 11891.705,E2 11891.705} C_VEL
LIN {X 0,Y 451.905,Z 777.899,A -85,B 0,C 180,E1 11891.237,E2 11891.237} C_VEL
LIN {X 0,Y 452.491,Z 770.376,A -85,B 0,C 180,E1 11891.004,E2 11891.004} C_VEL
LIN {X 0,Y 453.421,Z 750.849,A -85,B 0,C 180,E1 11889.952,E2 11889.952} C_VEL
LIN {X 0,Y 453.976,Z 744.378,A -85,B 0,C 180,E1 11889.766,E2 11889.766} C_VEL
LIN {X 0,Y 467.223,Z 620.542,A -85,B 0,C 180,E1 11888.027,E2 11888.027} C_VEL
LIN {X 0,Y 465.167,Z 616.161,A -85,B 0,C 180,E1 11885.18,E2 11885.18} C_VEL
LIN {X 0,Y 463.939,Z 612.005,A -85,B 0,C 180,E1 11880.617,E2 11880.617} C_VEL
LIN {X 0,Y 463.95,Z 612.34,A -85,B 0,C 180,E1 11879.259,E2 11879.259} C_VEL
LIN {X 0,Y 465.276,Z 616.26,A -85,B 0,C 180,E1 11875.069,E2 11875.069} C_VEL
LIN {X 0,Y 467.336,Z 620.867,A -85,B 0,C 180,E1 11872.253,E2 11872.253} C_VEL
LIN {X 0,Y 446.512,Z 814.448,A -85,B 0,C 180,E1 11869.549,E2 11869.549} C_VEL
LIN {X 0,Y 442.502,Z 839.948,A -85,B 0,C 180,E1 11869.151,E2 11869.151} C_VEL
LIN {X 0,Y 436.206,Z 868.173,A -85,B 0,C 180,E1 11868.647,E2 11868.647} C_VEL
LIN {X 0,Y 430.094,Z 890.12,A -85,B 0,C 180,E1 11868.157,E2 11868.157} C_VEL
LIN {X 0,Y 423.354,Z 910.794,A -85,B 0,C 180,E1 11867.589,E2 11867.589} C_VEL
LIN {X 0,Y 415.294,Z 932.315,A -85,B 0,C 180,E1 11866.873,E2 11866.873} C_VEL
LIN {X 0,Y 403.819,Z 958.875,A -85,B 0,C 180,E1 11865.778,E2 11865.778} C_VEL
LIN {X 0,Y 393.373,Z 979.947,A -85,B 0,C 180,E1 11864.708,E2 11864.708} C_VEL
LIN {X 0,Y 383.096,Z 998.757,A -85,B 0,C 180,E1 11863.567,E2 11863.567} C_VEL
LIN {X 0,Y 372.13,Z 1017.082,A -85,B 0,C 180,E1 11862.267,E2 11862.267} C_VEL
LIN {X 0,Y 358.98,Z 1037.303,A -85,B 0,C 180,E1 11860.547,E2 11860.547} C_VEL
LIN {X 0,Y 343.361,Z 1059.025,A -85,B 0,C 180,E1 11858.267,E2 11858.267} C_VEL
LIN {X 0,Y 330.643,Z 1075.378,A -85,B 0,C 180,E1 11856.17,E2 11856.17} C_VEL
LIN {X 0,Y 318.406,Z 1090.191,A -85,B 0,C 180,E1 11853.909,E2 11853.909} C_VEL
LIN {X 0,Y 305.651,Z 1104.81,A -85,B 0,C 180,E1 11851.245,E2 11851.245} C_VEL
LIN {X 0,Y 290.256,Z 1121.568,A -85,B 0,C 180,E1 11847.493,E2 11847.493} C_VEL
LIN {X 0,Y 276.953,Z 1135.281,A -85,B 0,C 180,E1 11843.617,E2 11843.617} C_VEL
LIN {X 0,Y 265.903,Z 1146.452,A -85,B 0,C 180,E1 11839.758,E2 11839.758} C_VEL
LIN {X 0,Y 256.047,Z 1156.354,A -85,B 0,C 180,E1 11835.611,E2 11835.611} C_VEL
LIN {X 0,Y 245.552,Z 1167.145,A -85,B 0,C 180,E1 11830.043,E2 11830.043} C_VEL
LIN {X 0,Y 236.899,Z 1176.321,A -85,B 0,C 180,E1 11823.857,E2 11823.857} C_VEL
LIN {X 0,Y 231.639,Z 1182.499,A -85,B 0,C 180,E1 11818.628,E2 11818.628} C_VEL
LIN {X 0,Y 227.904,Z 1187.574,A -85,B 0,C 180,E1 11813.256,E2 11813.256} C_VEL
LIN {X 0,Y 225.629,Z 1191.403,A -85,B 0,C 180,E1 11808.071,E2 11808.071} C_VEL
LIN {X 0,Y 224.465,Z 1194.149,A -85,B 0,C 180,E1 11803.131,E2 11803.131} C_VEL
LIN {X 0,Y 224.058,Z 1196.037,A -85,B 0,C 180,E1 11798.21,E2 11798.21} C_VEL
LIN {X 0,Y 224.012,Z 1197.042,A -85,B 0,C 180,E1 11793.583,E2 11793.583} C_VEL
LIN {X 0,Y 224.027,Z 1197.256,A -85,B 0,C 180,E1 11788.721,E2 11788.721} C_VEL
LIN {X 0,Y 224.016,Z 1196.533,A -85,B 0,C 180,E1 11783.593,E2 11783.593} C_VEL
LIN {X 0,Y 224.296,Z 1194.733,A -85,B 0,C 180,E1 11778.167,E2 11778.167} C_VEL
LIN {X 0,Y 225.39,Z 1191.885,A -85,B 0,C 180,E1 11772.709,E2 11772.709} C_VEL
LIN {X 0,Y 227.614,Z 1187.979,A -85,B 0,C 180,E1 11767.259,E2 11767.259} C_VEL
LIN {X 0,Y 231.217,Z 1182.996,A -85,B 0,C 180,E1 11761.878,E2 11761.878} C_VEL
LIN {X 0,Y 236.329,Z 1176.907,A -85,B 0,C 180,E1 11756.633,E2 11756.633} C_VEL
LIN {X 0,Y 243.696,Z 1168.948,A -85,B 0,C 180,E1 11751.116,E2 11751.116} C_VEL
LIN {X 0,Y 255.134,Z 1157.233,A -85,B 0,C 180,E1 11744.82,E2 11744.82} C_VEL
LIN {X 0,Y 265.374,Z 1146.909,A -85,B 0,C 180,E1 11740.441,E2 11740.441} C_VEL
LIN {X 0,Y 275.839,Z 1136.315,A -85,B 0,C 180,E1 11736.735,E2 11736.735} C_VEL
LIN {X 0,Y 287.822,Z 1123.939,A -85,B 0,C 180,E1 11733.154,E2 11733.154} C_VEL
LIN {X 0,Y 303.579,Z 1107.029,A -85,B 0,C 180,E1 11729.215,E2 11729.215} C_VEL
LIN {X 0,Y 317.667,Z 1090.901,A -85,B 0,C 180,E1 11726.229,E2 11726.229} C_VEL
LIN {X 0,Y 329.781,Z 1076.265,A -85,B 0,C 180,E1 11723.972,E2 11723.972} C_VEL
LIN {X 0,Y 342.168,Z 1060.378,A -85,B 0,C 180,E1 11721.91,E2 11721.91} C_VEL
LIN {X 0,Y 356.911,Z 1040.136,A -85,B 0,C 180,E1 11719.733,E2 11719.733} C_VEL
LIN {X 0,Y 371.283,Z 1018.161,A -85,B 0,C 180,E1 11717.831,E2 11717.831} C_VEL
LIN {X 0,Y 382.232,Z 999.935,A -85,B 0,C 180,E1 11716.524,E2 11716.524} C_VEL
LIN {X 0,Y 392.495,Z 981.244,A -85,B 0,C 180,E1 11715.377,E2 11715.377} C_VEL
LIN {X 0,Y 402.927,Z 960.318,A -85,B 0,C 180,E1 11714.299,E2 11714.299} C_VEL
LIN {X 0,Y 414.559,Z 933.69,A -85,B 0,C 180,E1 11713.186,E2 11713.186} C_VEL
LIN {X 0,Y 422.873,Z 911.586,A -85,B 0,C 180,E1 11712.443,E2 11712.443} C_VEL
LIN {X 0,Y 429.627,Z 890.965,A -85,B 0,C 180,E1 11711.871,E2 11711.871} C_VEL
LIN {X 0,Y 435.609,Z 869.644,A -85,B 0,C 180,E1 11711.39,E2 11711.39} C_VEL
LIN {X 0,Y 441.669,Z 843.319,A -85,B 0,C 180,E1 11710.909,E2 11710.909} C_VEL
LIN {X 0,Y 446.144,Z 815.621,A -85,B 0,C 180,E1 11710.473,E2 11710.473} C_VEL
LIN {X 0,Y 456.575,Z 719.136,A -85,B 0,C 180,E1 11709.115,E2 11709.115} C_VEL
LIN {X 0,Y 467.11,Z 620.507,A -85,B 0,C 180,E1 11707.719,E2 11707.719} C_VEL
LIN {X 0,Y 465.043,Z 616.084,A -85,B 0,C 180,E1 11704.934,E2 11704.934} C_VEL
LIN {X 0,Y 463.727,Z 612.363,A -85,B 0,C 180,E1 11701.112,E2 11701.112} C_VEL
LIN {X 0,Y 463.66,Z 611.979,A -85,B 0,C 180,E1 11700.247,E2 11700.247} C_VEL
LIN {X 0,Y 463.708,Z 612.146,A -85,B 0,C 180,E1 11698.641,E2 11698.641} C_VEL
LIN {X 0,Y 465.366,Z 616.872,A -85,B 0,C 180,E1 11694.018,E2 11694.018} C_VEL
LIN {X 0,Y 467.021,Z 620.505,A -85,B 0,C 180,E1 11691.853,E2 11691.853} C_VEL
LIN {X 0,Y 446.684,Z 809.093,A -85,B 0,C 180,E1 11689.227,E2 11689.227} C_VEL
LIN {X 0,Y 442.637,Z 834.698,A -85,B 0,C 180,E1 11688.829,E2 11688.829} C_VEL
LIN {X 0,Y 436.477,Z 862.478,A -85,B 0,C 180,E1 11688.279,E2 11688.279} C_VEL
LIN {X 0,Y 430.514,Z 884.115,A -85,B 0,C 180,E1 11687.736,E2 11687.736} C_VEL
LIN {X 0,Y 424.085,Z 904.026,A -85,B 0,C 180,E1 11687.135,E2 11687.135} C_VEL
LIN {X 0,Y 416.392,Z 924.78,A -85,B 0,C 180,E1 11686.389,E2 11686.389} C_VEL
LIN {X 0,Y 406.156,Z 948.997,A -85,B 0,C 180,E1 11685.345,E2 11685.345} C_VEL
LIN {X 0,Y 394.599,Z 972.443,A -85,B 0,C 180,E1 11684.096,E2 11684.096} C_VEL
LIN {X 0,Y 384.146,Z 991.493,A -85,B 0,C 180,E1 11682.895,E2 11682.895} C_VEL
LIN {X 0,Y 373.17,Z 1009.761,A -85,B 0,C 180,E1 11681.53,E2 11681.53} C_VEL
LIN {X 0,Y 360.966,Z 1028.391,A -85,B 0,C 180,E1 11679.886,E2 11679.886} C_VEL
LIN {X 0,Y 345.15,Z 1050.236,A -85,B 0,C 180,E1 11677.533,E2 11677.533} C_VEL
LIN {X 0,Y 332.931,Z 1065.738,A -85,B 0,C 180,E1 11675.501,E2 11675.501} C_VEL
LIN {X 0,Y 321.132,Z 1079.778,A -85,B 0,C 180,E1 11673.327,E2 11673.327} C_VEL
LIN {X 0,Y 308.435,Z 1094.039,A -85,B 0,C 180,E1 11670.694,E2 11670.694} C_VEL
LIN {X 0,Y 293.845,Z 1109.613,A -85,B 0,C 180,E1 11667.188,E2 11667.188} C_VEL
LIN {X 0,Y 279.187,Z 1124.218,A -85,B 0,C 180,E1 11663,E2 11663} C_VEL
LIN {X 0,Y 268.391,Z 1134.656,A -85,B 0,C 180,E1 11659.31,E2 11659.31} C_VEL
LIN {X 0,Y 258.341,Z 1144.195,A -85,B 0,C 180,E1 11655.217,E2 11655.217} C_VEL
LIN {X 0,Y 247.88,Z 1154.211,A -85,B 0,C 180,E1 11649.892,E2 11649.892} C_VEL
LIN {X 0,Y 238.563,Z 1163.254,A -85,B 0,C 180,E1 11643.589,E2 11643.589} C_VEL
LIN {X 0,Y 232.812,Z 1169.273,A -85,B 0,C 180,E1 11638.191,E2 11638.191} C_VEL
LIN {X 0,Y 228.803,Z 1173.931,A -85,B 0,C 180,E1 11632.888,E2 11632.888} C_VEL
LIN {X 0,Y 226.185,Z 1177.555,A -85,B 0,C 180,E1 11627.493,E2 11627.493} C_VEL
LIN {X 0,Y 224.744,Z 1180.181,A -85,B 0,C 180,E1 11622.069,E2 11622.069} C_VEL
LIN {X 0,Y 224.183,Z 1181.774,A -85,B 0,C 180,E1 11616.916,E2 11616.916} C_VEL
LIN {X 0,Y 224.035,Z 1182.484,A -85,B 0,C 180,E1 11612.046,E2 11612.046} C_VEL
LIN {X 0,Y 224.035,Z 1182.474,A -85,B 0,C 180,E1 11607.698,E2 11607.698} C_VEL
LIN {X 0,Y 224.176,Z 1181.806,A -85,B 0,C 180,E1 11603.083,E2 11603.083} C_VEL
LIN {X 0,Y 224.728,Z 1180.234,A -85,B 0,C 180,E1 11597.93,E2 11597.93} C_VEL
LIN {X 0,Y 226.155,Z 1177.629,A -85,B 0,C 180,E1 11592.504,E2 11592.504} C_VEL
LIN {X 0,Y 228.756,Z 1174.024,A -85,B 0,C 180,E1 11587.107,E2 11587.107} C_VEL
LIN {X 0,Y 232.851,Z 1169.269,A -85,B 0,C 180,E1 11581.678,E2 11581.678} C_VEL
LIN {X 0,Y 238.774,Z 1163.097,A -85,B 0,C 180,E1 11576.156,E2 11576.156} C_VEL
LIN {X 0,Y 248.541,Z 1153.603,A -85,B 0,C 180,E1 11569.633,E2 11569.633} C_VEL
LIN {X 0,Y 258.499,Z 1144.119,A -85,B 0,C 180,E1 11564.627,E2 11564.627} C_VEL
LIN {X 0,Y 268.499,Z 1134.636,A -85,B 0,C 180,E1 11560.565,E2 11560.565} C_VEL
LIN {X 0,Y 280.208,Z 1123.332,A -85,B 0,C 180,E1 11556.596,E2 11556.596} C_VEL
LIN {X 0,Y 296.264,Z 1107.15,A -85,B 0,C 180,E1 11552.103,E2 11552.103} C_VEL
LIN {X 0,Y 308.975,Z 1093.598,A -85,B 0,C 180,E1 11549.105,E2 11549.105} C_VEL
LIN {X 0,Y 320.984,Z 1080.121,A -85,B 0,C 180,E1 11546.62,E2 11546.62} C_VEL
LIN {X 0,Y 333.535,Z 1065.195,A -85,B 0,C 180,E1 11544.312,E2 11544.312} C_VEL
LIN {X 0,Y 348.521,Z 1046.111,A -85,B 0,C 180,E1 11541.864,E2 11541.864} C_VEL
LIN {X 0,Y 362.436,Z 1026.461,A -85,B 0,C 180,E1 11539.827,E2 11539.827} C_VEL
LIN {X 0,Y 373.862,Z 1008.96,A -85,B 0,C 180,E1 11538.303,E2 11538.303} C_VEL
LIN {X 0,Y 384.682,Z 990.908,A -85,B 0,C 180,E1 11536.963,E2 11536.963} C_VEL
LIN {X 0,Y 395.711,Z 970.725,A -85,B 0,C 180,E1 11535.702,E2 11535.702} C_VEL
LIN {X 0,Y 408.196,Z 944.748,A -85,B 0,C 180,E1 11534.36,E2 11534.36} C_VEL
LIN {X 0,Y 416.971,Z 923.825,A -85,B 0,C 180,E1 11533.476,E2 11533.476} C_VEL
LIN {X 0,Y 424.415,Z 903.683,A -85,B 0,C 180,E1 11532.756,E2 11532.756} C_VEL
LIN {X 0,Y 431.072,Z 882.975,A -85,B 0,C 180,E1 11532.136,E2 11532.136} C_VEL
LIN {X 0,Y 438,Z 857.453,A -85,B 0,C 180,E1 11531.513,E2 11531.513} C_VEL
LIN {X 0,Y 443.622,Z 830.231,A -85,B 0,C 180,E1 11531.003,E2 11531.003} C_VEL
LIN {X 0,Y 447.099,Z 807.568,A -85,B 0,C 180,E1 11530.656,E2 11530.656} C_VEL
LIN {X 0,Y 453.976,Z 744.378,A -85,B 0,C 180,E1 11529.766,E2 11529.766} C_VEL
LIN {X 0,Y 454.606,Z 736.858,A -85,B 0,C 180,E1 11529.534,E2 11529.534} C_VEL
LIN {X 0,Y 455.742,Z 717.344,A -85,B 0,C 180,E1 11528.487,E2 11528.487} C_VEL
LIN {X 0,Y 456.334,Z 710.874,A -85,B 0,C 180,E1 11528.303,E2 11528.303} C_VEL
LIN {X 0,Y 465.484,Z 627.17,A -85,B 0,C 180,E1 11527.157,E2 11527.157} C_VEL
LIN {X 0,Y 464.117,Z 624.043,A -85,B 0,C 180,E1 11525.068,E2 11525.068} C_VEL
LIN {X 0,Y 462.957,Z 619.954,A -85,B 0,C 180,E1 11520.495,E2 11520.495} C_VEL
LIN {X 0,Y 462.966,Z 620.351,A -85,B 0,C 180,E1 11519.258,E2 11519.258} C_VEL
LIN {X 0,Y 464.505,Z 624.844,A -85,B 0,C 180,E1 11514.689,E2 11514.689} C_VEL
LIN {X 0,Y 465.565,Z 627.472,A -85,B 0,C 180,E1 11513.142,E2 11513.142} C_VEL
LIN {X 0,Y 445.124,Z 814.189,A -85,B 0,C 180,E1 11510.569,E2 11510.569} C_VEL
LIN {X 0,Y 441.057,Z 839.7,A -85,B 0,C 180,E1 11510.179,E2 11510.179} C_VEL
LIN {X 0,Y 434.678,Z 867.967,A -85,B 0,C 180,E1 11509.687,E2 11509.687} C_VEL
LIN {X 0,Y 428.509,Z 889.864,A -85,B 0,C 180,E1 11509.214,E2 11509.214} C_VEL
LIN {X 0,Y 421.668,Z 910.589,A -85,B 0,C 180,E1 11508.662,E2 11508.662} C_VEL
LIN {X 0,Y 413.524,Z 932.055,A -85,B 0,C 180,E1 11507.969,E2 11507.969} C_VEL
LIN {X 0,Y 402.026,Z 958.339,A -85,B 0,C 180,E1 11506.919,E2 11506.919} C_VEL
LIN {X 0,Y 391.176,Z 979.898,A -85,B 0,C 180,E1 11505.853,E2 11505.853} C_VEL
LIN {X 0,Y 380.85,Z 998.491,A -85,B 0,C 180,E1 11504.754,E2 11504.754} C_VEL
LIN {X 0,Y 369.909,Z 1016.48,A -85,B 0,C 180,E1 11503.511,E2 11503.511} C_VEL
LIN {X 0,Y 356.903,Z 1036.15,A -85,B 0,C 180,E1 11501.882,E2 11501.882} C_VEL
LIN {X 0,Y 340.768,Z 1058.242,A -85,B 0,C 180,E1 11499.628,E2 11499.628} C_VEL
LIN {X 0,Y 327.357,Z 1075.107,A -85,B 0,C 180,E1 11497.508,E2 11497.508} C_VEL
LIN {X 0,Y 314.806,Z 1089.918,A -85,B 0,C 180,E1 11495.28,E2 11495.28} C_VEL
LIN {X 0,Y 301.692,Z 1104.536,A -85,B 0,C 180,E1 11492.647,E2 11492.647} C_VEL
LIN {X 0,Y 285.273,Z 1121.822,A -85,B 0,C 180,E1 11488.782,E2 11488.782} C_VEL
LIN {X 0,Y 271.796,Z 1135.232,A -85,B 0,C 180,E1 11484.977,E2 11484.977} C_VEL
LIN {X 0,Y 260.522,Z 1146.176,A -85,B 0,C 180,E1 11481.178,E2 11481.178} C_VEL
LIN {X 0,Y 249.722,Z 1156.548,A -85,B 0,C 180,E1 11476.778,E2 11476.778} C_VEL
LIN {X 0,Y 238.363,Z 1167.629,A -85,B 0,C 180,E1 11470.872,E2 11470.872} C_VEL
LIN {X 0,Y 229.669,Z 1176.36,A -85,B 0,C 180,E1 11464.771,E2 11464.771} C_VEL
LIN {X 0,Y 224.118,Z 1182.49,A -85,B 0,C 180,E1 11459.389,E2 11459.389} C_VEL
LIN {X 0,Y 220.154,Z 1187.518,A -85,B 0,C 180,E1 11453.841,E2 11453.841} C_VEL
LIN {X 0,Y 217.644,Z 1191.468,A -85,B 0,C 180,E1 11448.203,E2 11448.203} C_VEL
LIN {X 0,Y 216.412,Z 1194.241,A -85,B 0,C 180,E1 11442.813,E2 11442.813} C_VEL
LIN {X 0,Y 216.048,Z 1195.99,A -85,B 0,C 180,E1 11437.713,E2 11437.713} C_VEL
LIN {X 0,Y 216.019,Z 1196.828,A -85,B 0,C 180,E1 11433.184,E2 11433.184} C_VEL
LIN {X 0,Y 216.031,Z 1196.994,A -85,B 0,C 180,E1 11428.674,E2 11428.674} C_VEL
LIN {X 0,Y 216.018,Z 1196.34,A -85,B 0,C 180,E1 11423.622,E2 11423.622} C_VEL
LIN {X 0,Y 216.311,Z 1194.586,A -85,B 0,C 180,E1 11417.995,E2 11417.995} C_VEL
LIN {X 0,Y 217.565,Z 1191.607,A -85,B 0,C 180,E1 11412.053,E2 11412.053} C_VEL
LIN {X 0,Y 220.002,Z 1187.707,A -85,B 0,C 180,E1 11406.426,E2 11406.426} C_VEL
LIN {X 0,Y 223.889,Z 1182.721,A -85,B 0,C 180,E1 11400.871,E2 11400.871} C_VEL
LIN {X 0,Y 229.365,Z 1176.631,A -85,B 0,C 180,E1 11395.48,E2 11395.48} C_VEL
LIN {X 0,Y 237.507,Z 1168.369,A -85,B 0,C 180,E1 11389.641,E2 11389.641} C_VEL
LIN {X 0,Y 249.238,Z 1156.953,A -85,B 0,C 180,E1 11383.439,E2 11383.439} C_VEL
LIN {X 0,Y 259.966,Z 1146.63,A -85,B 0,C 180,E1 11379.021,E2 11379.021} C_VEL
LIN {X 0,Y 270.815,Z 1136.09,A -85,B 0,C 180,E1 11375.32,E2 11375.32} C_VEL
LIN {X 0,Y 283.295,Z 1123.66,A -85,B 0,C 180,E1 11371.725,E2 11371.725} C_VEL
LIN {X 0,Y 299.563,Z 1106.75,A -85,B 0,C 180,E1 11367.811,E2 11367.811} C_VEL
LIN {X 0,Y 314.084,Z 1090.582,A -85,B 0,C 180,E1 11364.849,E2 11364.849} C_VEL
LIN {X 0,Y 326.568,Z 1075.874,A -85,B 0,C 180,E1 11362.616,E2 11362.616} C_VEL
LIN {X 0,Y 339.148,Z 1060.101,A -85,B 0,C 180,E1 11360.604,E2 11360.604} C_VEL
LIN {X 0,Y 354.194,Z 1039.861,A -85,B 0,C 180,E1 11358.469,E2 11358.469} C_VEL
LIN {X 0,Y 368.836,Z 1017.885,A -85,B 0,C 180,E1 11356.608,E2 11356.608} C_VEL
LIN {X 0,Y 379.972,Z 999.66,A -85,B 0,C 180,E1 11355.333,E2 11355.333} C_VEL
LIN {X 0,Y 390.138,Z 981.462,A -85,B 0,C 180,E1 11354.243,E2 11354.243} C_VEL
LIN {X 0,Y 400.099,Z 961.856,A -85,B 0,C 180,E1 11353.253,E2 11353.253} C_VEL
LIN {X 0,Y 411.268,Z 937.25,A -85,B 0,C 180,E1 11352.225,E2 11352.225} C_VEL
LIN {X 0,Y 420.747,Z 912.602,A -85,B 0,C 180,E1 11351.404,E2 11351.404} C_VEL
LIN {X 0,Y 427.809,Z 891.433,A -85,B 0,C 180,E1 11350.831,E2 11350.831} C_VEL
LIN {X 0,Y 433.831,Z 870.344,A -85,B 0,C 180,E1 11350.366,E2 11350.366} C_VEL
LIN {X 0,Y 439.336,Z 847.041,A -85,B 0,C 180,E1 11349.948,E2 11349.948} C_VEL
LIN {X 0,Y 444.551,Z 816.884,A -85,B 0,C 180,E1 11349.475,E2 11349.475} C_VEL
LIN {X 0,Y 451.654,Z 753.314,A -85,B 0,C 180,E1 11348.587,E2 11348.587} C_VEL
LIN {X 0,Y 465.356,Z 627.155,A -85,B 0,C 180,E1 11346.855,E2 11346.855} C_VEL
LIN {X 0,Y 463.914,Z 623.864,A -85,B 0,C 180,E1 11344.698,E2 11344.698} C_VEL
LIN {X 0,Y 462.735,Z 620.093,A -85,B 0,C 180,E1 11340.867,E2 11340.867} C_VEL
LIN {X 0,Y 462.723,Z 620.027,A -85,B 0,C 180,E1 11338.762,E2 11338.762} C_VEL
LIN {X 0,Y 464.265,Z 624.675,A -85,B 0,C 180,E1 11334.19,E2 11334.19} C_VEL
LIN {X 0,Y 465.242,Z 627.243,A -85,B 0,C 180,E1 11332.741,E2 11332.741} C_VEL
LIN {X 0,Y 445.257,Z 809.377,A -85,B 0,C 180,E1 11330.239,E2 11330.239} C_VEL
LIN {X 0,Y 441.155,Z 834.978,A -85,B 0,C 180,E1 11329.849,E2 11329.849} C_VEL
LIN {X 0,Y 434.947,Z 862.644,A -85,B 0,C 180,E1 11329.316,E2 11329.316} C_VEL
LIN {X 0,Y 428.879,Z 884.388,A -85,B 0,C 180,E1 11328.784,E2 11328.784} C_VEL
LIN {X 0,Y 422.366,Z 904.298,A -85,B 0,C 180,E1 11328.2,E2 11328.2} C_VEL
LIN {X 0,Y 414.783,Z 924.507,A -85,B 0,C 180,E1 11327.494,E2 11327.494} C_VEL
LIN {X 0,Y 405.061,Z 947.274,A -85,B 0,C 180,E1 11326.545,E2 11326.545} C_VEL
LIN {X 0,Y 392.84,Z 971.991,A -85,B 0,C 180,E1 11325.279,E2 11325.279} C_VEL
LIN {X 0,Y 382.151,Z 991.218,A -85,B 0,C 180,E1 11324.099,E2 11324.099} C_VEL
LIN {X 0,Y 371.506,Z 1008.711,A -85,B 0,C 180,E1 11322.83,E2 11322.83} C_VEL
LIN {X 0,Y 360.174,Z 1025.807,A -85,B 0,C 180,E1 11321.382,E2 11321.382} C_VEL
LIN {X 0,Y 346.07,Z 1045.402,A -85,B 0,C 180,E1 11319.405,E2 11319.405} C_VEL
LIN {X 0,Y 330.358,Z 1065.099,A -85,B 0,C 180,E1 11316.938,E2 11316.938} C_VEL
LIN {X 0,Y 317.28,Z 1080.301,A -85,B 0,C 180,E1 11314.621,E2 11314.621} C_VEL
LIN {X 0,Y 304.457,Z 1094.315,A -85,B 0,C 180,E1 11312.057,E2 11312.057} C_VEL
LIN {X 0,Y 289.274,Z 1110.039,A -85,B 0,C 180,E1 11308.537,E2 11308.537} C_VEL
LIN {X 0,Y 274.246,Z 1124.494,A -85,B 0,C 180,E1 11304.392,E2 11304.392} C_VEL
LIN {X 0,Y 262.73,Z 1135.201,A -85,B 0,C 180,E1 11300.583,E2 11300.583} C_VEL
LIN {X 0,Y 252.346,Z 1144.646,A -85,B 0,C 180,E1 11296.476,E2 11296.476} C_VEL
LIN {X 0,Y 241.133,Z 1154.88,A -85,B 0,C 180,E1 11290.931,E2 11290.931} C_VEL
LIN {X 0,Y 231.691,Z 1163.527,A -85,B 0,C 180,E1 11284.725,E2 11284.725} C_VEL
LIN {X 0,Y 225.506,Z 1169.595,A -85,B 0,C 180,E1 11279.132,E2 11279.132} C_VEL
LIN {X 0,Y 221.249,Z 1174.201,A -85,B 0,C 180,E1 11273.716,E2 11273.716} C_VEL
LIN {X 0,Y 218.408,Z 1177.823,A -85,B 0,C 180,E1 11268.138,E2 11268.138} C_VEL
LIN {X 0,Y 216.823,Z 1180.448,A -85,B 0,C 180,E1 11262.517,E2 11262.517} C_VEL
LIN {X 0,Y 216.203,Z 1182.038,A -85,B 0,C 180,E1 11257.173,E2 11257.173} C_VEL
LIN {X 0,Y 216.039,Z 1182.747,A -85,B 0,C 180,E1 11252.122,E2 11252.122} C_VEL
LIN {X 0,Y 216.04,Z 1182.736,A -85,B 0,C 180,E1 11247.613,E2 11247.613} C_VEL
LIN {X 0,Y 216.198,Z 1182.069,A -85,B 0,C 180,E1 11242.827,E2 11242.827} C_VEL
LIN {X 0,Y 216.806,Z 1180.5,A -85,B 0,C 180,E1 11237.482,E2 11237.482} C_VEL
LIN {X 0,Y 218.374,Z 1177.896,A -85,B 0,C 180,E1 11231.86,E2 11231.86} C_VEL
LIN {X 0,Y 221.201,Z 1174.294,A -85,B 0,C 180,E1 11226.279,E2 11226.279} C_VEL
LIN {X 0,Y 225.484,Z 1169.658,A -85,B 0,C 180,E1 11220.806,E2 11220.806} C_VEL
LIN {X 0,Y 231.597,Z 1163.662,A -85,B 0,C 180,E1 11215.259,E2 11215.259} C_VEL
LIN {X 0,Y 241.079,Z 1155.001,A -85,B 0,C 180,E1 11209.013,E2 11209.013} C_VEL
LIN {X 0,Y 252.219,Z 1144.839,A -85,B 0,C 180,E1 11203.493,E2 11203.493} C_VEL
LIN {X 0,Y 262.595,Z 1135.412,A -85,B 0,C 180,E1 11199.381,E2 11199.381} C_VEL
LIN {X 0,Y 274.104,Z 1124.727,A -85,B 0,C 180,E1 11195.566,E2 11195.566} C_VEL
LIN {X 0,Y 288.646,Z 1110.788,A -85,B 0,C 180,E1 11191.539,E2 11191.539} C_VEL
LIN {X 0,Y 303.609,Z 1095.384,A -85,B 0,C 180,E1 11188.044,E2 11188.044} C_VEL
LIN {X 0,Y 316.618,Z 1081.223,A -85,B 0,C 180,E1 11185.423,E2 11185.423} C_VEL
LIN {X 0,Y 329.449,Z 1066.376,A -85,B 0,C 180,E1 11183.135,E2 11183.135} C_VEL
LIN {X 0,Y 342.747,Z 1049.902,A -85,B 0,C 180,E1 11181.013,E2 11181.013} C_VEL
LIN {X 0,Y 358.917,Z 1027.93,A -85,B 0,C 180,E1 11178.71,E2 11178.71} C_VEL
LIN {X 0,Y 370.958,Z 1009.885,A -85,B 0,C 180,E1 11177.158,E2 11177.158} C_VEL
LIN {X 0,Y 381.957,Z 991.898,A -85,B 0,C 180,E1 11175.844,E2 11175.844} C_VEL
LIN {X 0,Y 392.29,Z 973.401,A -85,B 0,C 180,E1 11174.703,E2 11174.703} C_VEL
LIN {X 0,Y 403.629,Z 950.856,A -85,B 0,C 180,E1 11173.521,E2 11173.521} C_VEL
LIN {X 0,Y 414.232,Z 926.442,A -85,B 0,C 180,E1 11172.482,E2 11172.482} C_VEL
LIN {X 0,Y 421.996,Z 905.979,A -85,B 0,C 180,E1 11171.758,E2 11171.758} C_VEL
LIN {X 0,Y 428.756,Z 885.512,A -85,B 0,C 180,E1 11171.149,E2 11171.149} C_VEL
LIN {X 0,Y 434.792,Z 864.079,A -85,B 0,C 180,E1 11170.62,E2 11170.62} C_VEL
LIN {X 0,Y 440.752,Z 838.3,A -85,B 0,C 180,E1 11170.112,E2 11170.112} C_VEL
LIN {X 0,Y 445.328,Z 810.586,A -85,B 0,C 180,E1 11169.684,E2 11169.684} C_VEL
LIN {X 0,Y 455.351,Z 719.944,A -85,B 0,C 180,E1 11168.427,E2 11168.427} C_VEL
LIN {X 0,Y 456.334,Z 710.874,A -85,B 0,C 180,E1 11168.303,E2 11168.303} C_VEL
LIN {X 0,Y 457.013,Z 703.353,A -85,B 0,C 180,E1 11168.075,E2 11168.075} C_VEL
LIN {X 0,Y 458.356,Z 683.845,A -85,B 0,C 180,E1 11167.035,E2 11167.035} C_VEL
LIN {X 0,Y 458.983,Z 677.376,A -85,B 0,C 180,E1 11166.852,E2 11166.852} C_VEL
LIN {X 0,Y 463.821,Z 633.853,A -85,B 0,C 180,E1 11166.25,E2 11166.25} C_VEL
LIN {X 0,Y 463,Z 631.828,A -85,B 0,C 180,E1 11164.831,E2 11164.831} C_VEL
LIN {X 0,Y 461.982,Z 627.895,A -85,B 0,C 180,E1 11160.496,E2 11160.496} C_VEL
LIN {X 0,Y 461.983,Z 628.228,A -85,B 0,C 180,E1 11159.38,E2 11159.38} C_VEL
LIN {X 0,Y 463.409,Z 632.645,A -85,B 0,C 180,E1 11154.863,E2 11154.863} C_VEL
LIN {X 0,Y 463.892,Z 634.197,A -85,B 0,C 180,E1 11154.035,E2 11154.035} C_VEL
LIN {X 0,Y 443.862,Z 814.049,A -85,B 0,C 180,E1 11151.593,E2 11151.593} C_VEL
LIN {X 0,Y 439.641,Z 840.103,A -85,B 0,C 180,E1 11151.202,E2 11151.202} C_VEL
LIN {X 0,Y 433.25,Z 867.931,A -85,B 0,C 180,E1 11150.732,E2 11150.732} C_VEL
LIN {X 0,Y 427.072,Z 889.608,A -85,B 0,C 180,E1 11150.278,E2 11150.278} C_VEL
LIN {X 0,Y 420.152,Z 910.33,A -85,B 0,C 180,E1 11149.745,E2 11149.745} C_VEL
LIN {X 0,Y 411.907,Z 931.794,A -85,B 0,C 180,E1 11149.075,E2 11149.075} C_VEL
LIN {X 0,Y 400.076,Z 958.441,A -85,B 0,C 180,E1 11148.041,E2 11148.041} C_VEL
LIN {X 0,Y 388.926,Z 980.236,A -85,B 0,C 180,E1 11146.991,E2 11146.991} C_VEL
LIN {X 0,Y 378.331,Z 998.967,A -85,B 0,C 180,E1 11145.909,E2 11145.909} C_VEL
LIN {X 0,Y 367.006,Z 1017.222,A -85,B 0,C 180,E1 11144.671,E2 11144.671} C_VEL
LIN {X 0,Y 352.09,Z 1039.248,A -85,B 0,C 180,E1 11142.859,E2 11142.859} C_VEL
LIN {X 0,Y 336.73,Z 1059.51,A -85,B 0,C 180,E1 11140.776,E2 11140.776} C_VEL
LIN {X 0,Y 323.856,Z 1075.305,A -85,B 0,C 180,E1 11138.809,E2 11138.809} C_VEL
LIN {X 0,Y 311.39,Z 1089.645,A -85,B 0,C 180,E1 11136.683,E2 11136.683} C_VEL
LIN {X 0,Y 297.914,Z 1104.262,A -85,B 0,C 180,E1 11134.087,E2 11134.087} C_VEL
LIN {X 0,Y 280.995,Z 1121.547,A -85,B 0,C 180,E1 11130.252,E2 11130.252} C_VEL
LIN {X 0,Y 267.284,Z 1134.73,A -85,B 0,C 180,E1 11126.532,E2 11126.532} C_VEL
LIN {X 0,Y 255.31,Z 1145.9,A -85,B 0,C 180,E1 11122.655,E2 11122.655} C_VEL
LIN {X 0,Y 244.009,Z 1156.272,A -85,B 0,C 180,E1 11118.225,E2 11118.225} C_VEL
LIN {X 0,Y 231.856,Z 1167.529,A -85,B 0,C 180,E1 11112.118,E2 11112.118} C_VEL
LIN {X 0,Y 222.823,Z 1176.085,A -85,B 0,C 180,E1 11106.003,E2 11106.003} C_VEL
LIN {X 0,Y 216.842,Z 1182.262,A -85,B 0,C 180,E1 11100.425,E2 11100.425} C_VEL
LIN {X 0,Y 212.591,Z 1187.246,A -85,B 0,C 180,E1 11094.745,E2 11094.745} C_VEL
LIN {X 0,Y 209.842,Z 1191.199,A -85,B 0,C 180,E1 11088.905,E2 11088.905} C_VEL
LIN {X 0,Y 208.458,Z 1194.036,A -85,B 0,C 180,E1 11083.166,E2 11083.166} C_VEL
LIN {X 0,Y 208.051,Z 1195.797,A -85,B 0,C 180,E1 11077.733,E2 11077.733} C_VEL
LIN {X 0,Y 208.023,Z 1196.59,A -85,B 0,C 180,E1 11073.031,E2 11073.031} C_VEL
LIN {X 0,Y 208.033,Z 1196.708,A -85,B 0,C 180,E1 11068.348,E2 11068.348} C_VEL
LIN {X 0,Y 208.03,Z 1196.005,A -85,B 0,C 180,E1 11063.099,E2 11063.099} C_VEL
LIN {X 0,Y 208.398,Z 1194.198,A -85,B 0,C 180,E1 11057.25,E2 11057.25} C_VEL
LIN {X 0,Y 209.75,Z 1191.345,A -85,B 0,C 180,E1 11051.374,E2 11051.374} C_VEL
LIN {X 0,Y 212.427,Z 1187.434,A -85,B 0,C 180,E1 11045.531,E2 11045.531} C_VEL
LIN {X 0,Y 216.637,Z 1182.447,A -85,B 0,C 180,E1 11039.796,E2 11039.796} C_VEL
LIN {X 0,Y 222.498,Z 1176.354,A -85,B 0,C 180,E1 11034.254,E2 11034.254} C_VEL
LIN {X 0,Y 231.221,Z 1168.028,A -85,B 0,C 180,E1 11028.246,E2 11028.246} C_VEL
LIN {X 0,Y 243.499,Z 1156.674,A -85,B 0,C 180,E1 11021.994,E2 11021.994} C_VEL
LIN {X 0,Y 254.731,Z 1146.351,A -85,B 0,C 180,E1 11017.545,E2 11017.545} C_VEL
LIN {X 0,Y 266.263,Z 1135.586,A -85,B 0,C 180,E1 11013.765,E2 11013.765} C_VEL
LIN {X 0,Y 278.952,Z 1123.382,A -85,B 0,C 180,E1 11010.251,E2 11010.251} C_VEL
LIN {X 0,Y 295.009,Z 1107.255,A -85,B 0,C 180,E1 11006.523,E2 11006.523} C_VEL
LIN {X 0,Y 309.881,Z 1091.171,A -85,B 0,C 180,E1 11003.585,E2 11003.585} C_VEL
LIN {X 0,Y 323.05,Z 1076.066,A -85,B 0,C 180,E1 11001.313,E2 11001.313} C_VEL
LIN {X 0,Y 335.898,Z 1060.338,A -85,B 0,C 180,E1 10999.335,E2 10999.335} C_VEL
LIN {X 0,Y 349.969,Z 1041.83,A -85,B 0,C 180,E1 10997.402,E2 10997.402} C_VEL
LIN {X 0,Y 365.643,Z 1019.047,A -85,B 0,C 180,E1 10995.478,E2 10995.478} C_VEL
LIN {X 0,Y 377.441,Z 1000.127,A -85,B 0,C 180,E1 10994.176,E2 10994.176} C_VEL
LIN {X 0,Y 388.024,Z 981.514,A -85,B 0,C 180,E1 10993.088,E2 10993.088} C_VEL
LIN {X 0,Y 398.165,Z 961.865,A -85,B 0,C 180,E1 10992.121,E2 10992.121} C_VEL
LIN {X 0,Y 409.528,Z 937.205,A -85,B 0,C 180,E1 10991.121,E2 10991.121} C_VEL
LIN {X 0,Y 419.266,Z 912.199,A -85,B 0,C 180,E1 10990.315,E2 10990.315} C_VEL
LIN {X 0,Y 426.365,Z 891.159,A -85,B 0,C 180,E1 10989.764,E2 10989.764} C_VEL
LIN {X 0,Y 432.418,Z 870.199,A -85,B 0,C 180,E1 10989.317,E2 10989.317} C_VEL
LIN {X 0,Y 437.969,Z 846.98,A -85,B 0,C 180,E1 10988.914,E2 10988.914} C_VEL
LIN {X 0,Y 443.296,Z 816.598,A -85,B 0,C 180,E1 10988.448,E2 10988.448} C_VEL
LIN {X 0,Y 450.535,Z 752.897,A -85,B 0,C 180,E1 10987.572,E2 10987.572} C_VEL
LIN {X 0,Y 463.671,Z 633.8,A -85,B 0,C 180,E1 10985.941,E2 10985.941} C_VEL
LIN {X 0,Y 462.794,Z 631.643,A -85,B 0,C 180,E1 10984.461,E2 10984.461} C_VEL
LIN {X 0,Y 461.72,Z 627.86,A -85,B 0,C 180,E1 10980.372,E2 10980.372} C_VEL
LIN {X 0,Y 461.738,Z 628.052,A -85,B 0,C 180,E1 10978.759,E2 10978.759} C_VEL
LIN {X 0,Y 463.203,Z 632.585,A -85,B 0,C 180,E1 10974.301,E2 10974.301} C_VEL
LIN {X 0,Y 463.591,Z 633.846,A -85,B 0,C 180,E1 10973.636,E2 10973.636} C_VEL
LIN {X 0,Y 443.97,Z 809.662,A -85,B 0,C 180,E1 10971.257,E2 10971.257} C_VEL
LIN {X 0,Y 439.786,Z 835.419,A -85,B 0,C 180,E1 10970.873,E2 10970.873} C_VEL
LIN {X 0,Y 433.503,Z 863.026,A -85,B 0,C 180,E1 10970.355,E2 10970.355} C_VEL
LIN {X 0,Y 427.389,Z 884.661,A -85,B 0,C 180,E1 10969.841,E2 10969.841} C_VEL
LIN {X 0,Y 420.793,Z 904.57,A -85,B 0,C 180,E1 10969.273,E2 10969.273} C_VEL
LIN {X 0,Y 412.969,Z 925.134,A -85,B 0,C 180,E1 10968.573,E2 10968.573} C_VEL
LIN {X 0,Y 402.367,Z 949.541,A -85,B 0,C 180,E1 10967.575,E2 10967.575} C_VEL
LIN {X 0,Y 390.216,Z 973.432,A -85,B 0,C 180,E1 10966.365,E2 10966.365} C_VEL
LIN {X 0,Y 379.495,Z 992.339,A -85,B 0,C 180,E1 10965.225,E2 10965.225} C_VEL
LIN {X 0,Y 368.12,Z 1010.622,A -85,B 0,C 180,E1 10963.915,E2 10963.915} C_VEL
LIN {X 0,Y 354.829,Z 1030.141,A -85,B 0,C 180,E1 10962.257,E2 10962.257} C_VEL
LIN {X 0,Y 338.882,Z 1051.177,A -85,B 0,C 180,E1 10960.057,E2 10960.057} C_VEL
LIN {X 0,Y 326.425,Z 1066.286,A -85,B 0,C 180,E1 10958.141,E2 10958.141} C_VEL
LIN {X 0,Y 313.259,Z 1081.192,A -85,B 0,C 180,E1 10955.885,E2 10955.885} C_VEL
LIN {X 0,Y 299.209,Z 1096.105,A -85,B 0,C 180,E1 10953.154,E2 10953.154} C_VEL
LIN {X 0,Y 281.783,Z 1113.324,A -85,B 0,C 180,E1 10949.17,E2 10949.17} C_VEL
LIN {X 0,Y 268.851,Z 1125.331,A -85,B 0,C 180,E1 10945.651,E2 10945.651} C_VEL
LIN {X 0,Y 257.505,Z 1135.477,A -85,B 0,C 180,E1 10942.02,E2 10942.02} C_VEL
LIN {X 0,Y 246.681,Z 1144.921,A -85,B 0,C 180,E1 10937.88,E2 10937.88} C_VEL
LIN {X 0,Y 235.322,Z 1154.761,A -85,B 0,C 180,E1 10932.499,E2 10932.499} C_VEL
LIN {X 0,Y 224.912,Z 1163.801,A -85,B 0,C 180,E1 10925.931,E2 10925.931} C_VEL
LIN {X 0,Y 218.364,Z 1169.818,A -85,B 0,C 180,E1 10920.243,E2 10920.243} C_VEL
LIN {X 0,Y 213.742,Z 1174.472,A -85,B 0,C 180,E1 10914.603,E2 10914.603} C_VEL
LIN {X 0,Y 210.657,Z 1178.092,A -85,B 0,C 180,E1 10908.83,E2 10908.83} C_VEL
LIN {X 0,Y 208.911,Z 1180.714,A -85,B 0,C 180,E1 10903,E2 10903} C_VEL
LIN {X 0,Y 208.224,Z 1182.302,A -85,B 0,C 180,E1 10897.449,E2 10897.449} C_VEL
LIN {X 0,Y 208.046,Z 1182.988,A -85,B 0,C 180,E1 10892.479,E2 10892.479} C_VEL
LIN {X 0,Y 208.043,Z 1183.02,A -85,B 0,C 180,E1 10887.797,E2 10887.797} C_VEL
LIN {X 0,Y 208.218,Z 1182.333,A -85,B 0,C 180,E1 10882.55,E2 10882.55} C_VEL
LIN {X 0,Y 208.895,Z 1180.766,A -85,B 0,C 180,E1 10876.999,E2 10876.999} C_VEL
LIN {X 0,Y 210.62,Z 1178.164,A -85,B 0,C 180,E1 10871.167,E2 10871.167} C_VEL
LIN {X 0,Y 213.692,Z 1174.563,A -85,B 0,C 180,E1 10865.391,E2 10865.391} C_VEL
LIN {X 0,Y 218.289,Z 1169.929,A -85,B 0,C 180,E1 10859.745,E2 10859.745} C_VEL
LIN {X 0,Y 224.83,Z 1163.92,A -85,B 0,C 180,E1 10854.039,E2 10854.039} C_VEL
LIN {X 0,Y 234.781,Z 1155.33,A -85,B 0,C 180,E1 10847.711,E2 10847.711} C_VEL
LIN {X 0,Y 246.554,Z 1145.111,A -85,B 0,C 180,E1 10842.087,E2 10842.087} C_VEL
LIN {X 0,Y 257.797,Z 1135.309,A -85,B 0,C 180,E1 10837.794,E2 10837.794} C_VEL
LIN {X 0,Y 269.958,Z 1124.438,A -85,B 0,C 180,E1 10833.938,E2 10833.938} C_VEL
LIN {X 0,Y 285.709,Z 1109.756,A -85,B 0,C 180,E1 10829.786,E2 10829.786} C_VEL
LIN {X 0,Y 300.665,Z 1094.745,A -85,B 0,C 180,E1 10826.464,E2 10826.464} C_VEL
LIN {X 0,Y 313.909,Z 1080.66,A -85,B 0,C 180,E1 10823.915,E2 10823.915} C_VEL
LIN {X 0,Y 327.864,Z 1064.818,A -85,B 0,C 180,E1 10821.545,E2 10821.545} C_VEL
LIN {X 0,Y 344.763,Z 1043.904,A -85,B 0,C 180,E1 10819.014,E2 10819.014} C_VEL
LIN {X 0,Y 358.041,Z 1025.788,A -85,B 0,C 180,E1 10817.243,E2 10817.243} C_VEL
LIN {X 0,Y 369.249,Z 1009.193,A -85,B 0,C 180,E1 10815.873,E2 10815.873} C_VEL
LIN {X 0,Y 380.249,Z 991.433,A -85,B 0,C 180,E1 10814.614,E2 10814.614} C_VEL
LIN {X 0,Y 391.626,Z 971.247,A -85,B 0,C 180,E1 10813.412,E2 10813.412} C_VEL
LIN {X 0,Y 404.341,Z 945.593,A -85,B 0,C 180,E1 10812.154,E2 10812.154} C_VEL
LIN {X 0,Y 413.593,Z 924.127,A -85,B 0,C 180,E1 10811.293,E2 10811.293} C_VEL
LIN {X 0,Y 421.152,Z 904.196,A -85,B 0,C 180,E1 10810.619,E2 10810.619} C_VEL
LIN {X 0,Y 427.982,Z 883.484,A -85,B 0,C 180,E1 10810.032,E2 10810.032} C_VEL
LIN {X 0,Y 435.082,Z 857.958,A -85,B 0,C 180,E1 10809.442,E2 10809.442} C_VEL
LIN {X 0,Y 440.846,Z 830.724,A -85,B 0,C 180,E1 10808.959,E2 10808.959} C_VEL
LIN {X 0,Y 444.416,Z 808.05,A -85,B 0,C 180,E1 10808.626,E2 10808.626} C_VEL
LIN {X 0,Y 458.983,Z 677.376,A -85,B 0,C 180,E1 10806.852,E2 10806.852} C_VEL
LIN {X 0,Y 459.703,Z 669.86,A -85,B 0,C 180,E1 10806.624,E2 10806.624} C_VEL
LIN {X 0,Y 461.251,Z 650.366,A -85,B 0,C 180,E1 10805.591,E2 10805.591} C_VEL
LIN {X 0,Y 461.916,Z 643.899,A -85,B 0,C 180,E1 10805.413,E2 10805.413} C_VEL
LIN {X 0,Y 462.286,Z 640.446,A -85,B 0,C 180,E1 10805.337,E2 10805.337} C_VEL
LIN {X 0,Y 461.002,Z 635.843,A -85,B 0,C 180,E1 10800.373,E2 10800.373} C_VEL
LIN {X 0,Y 461,Z 636.236,A -85,B 0,C 180,E1 10799.379,E2 10799.379} C_VEL
LIN {X 0,Y 462.349,Z 640.554,A -85,B 0,C 180,E1 10794.975,E2 10794.975} C_VEL
LIN {X 0,Y 462.26,Z 641.569,A -85,B 0,C 180,E1 10794.927,E2 10794.927} C_VEL
LIN {X 0,Y 442.756,Z 813.806,A -85,B 0,C 180,E1 10792.624,E2 10792.624} C_VEL
LIN {X 0,Y 438.476,Z 839.887,A -85,B 0,C 180,E1 10792.242,E2 10792.242} C_VEL
LIN {X 0,Y 432.008,Z 867.74,A -85,B 0,C 180,E1 10791.785,E2 10791.785} C_VEL
LIN {X 0,Y 425.782,Z 889.352,A -85,B 0,C 180,E1 10791.349,E2 10791.349} C_VEL
LIN {X 0,Y 418.942,Z 909.641,A -85,B 0,C 180,E1 10790.847,E2 10790.847} C_VEL
LIN {X 0,Y 410.609,Z 931.128,A -85,B 0,C 180,E1 10790.202,E2 10790.202} C_VEL
LIN {X 0,Y 399.427,Z 956.276,A -85,B 0,C 180,E1 10789.269,E2 10789.269} C_VEL
LIN {X 0,Y 387.661,Z 979.073,A -85,B 0,C 180,E1 10788.219,E2 10788.219} C_VEL
LIN {X 0,Y 376.857,Z 997.961,A -85,B 0,C 180,E1 10787.169,E2 10787.169} C_VEL
LIN {X 0,Y 365.408,Z 1016.192,A -85,B 0,C 180,E1 10785.975,E2 10785.975} C_VEL
LIN {X 0,Y 352.316,Z 1035.315,A -85,B 0,C 180,E1 10784.469,E2 10784.469} C_VEL
LIN {X 0,Y 335.339,Z 1057.703,A -85,B 0,C 180,E1 10782.294,E2 10782.294} C_VEL
LIN {X 0,Y 321.742,Z 1074.095,A -85,B 0,C 180,E1 10780.324,E2 10780.324} C_VEL
LIN {X 0,Y 308.947,Z 1088.515,A -85,B 0,C 180,E1 10778.252,E2 10778.252} C_VEL
LIN {X 0,Y 295.834,Z 1102.422,A -85,B 0,C 180,E1 10775.859,E2 10775.859} C_VEL
LIN {X 0,Y 281.847,Z 1116.451,A -85,B 0,C 180,E1 10772.927,E2 10772.927} C_VEL
LIN {X 0,Y 264.024,Z 1133.284,A -85,B 0,C 180,E1 10768.438,E2 10768.438} C_VEL
LIN {X 0,Y 250.981,Z 1144.999,A -85,B 0,C 180,E1 10764.433,E2 10764.433} C_VEL
LIN {X 0,Y 239.533,Z 1155.055,A -85,B 0,C 180,E1 10760.179,E2 10760.179} C_VEL
LIN {X 0,Y 228.564,Z 1164.651,A -85,B 0,C 180,E1 10755.127,E2 10755.127} C_VEL
LIN {X 0,Y 217.001,Z 1174.982,A -85,B 0,C 180,E1 10748.007,E2 10748.007} C_VEL
LIN {X 0,Y 209.987,Z 1181.679,A -85,B 0,C 180,E1 10741.906,E2 10741.906} C_VEL
LIN {X 0,Y 205.261,Z 1186.758,A -85,B 0,C 180,E1 10736.002,E2 10736.002} C_VEL
LIN {X 0,Y 202.17,Z 1190.761,A -85,B 0,C 180,E1 10729.953,E2 10729.953} C_VEL
LIN {X 0,Y 200.656,Z 1193.467,A -85,B 0,C 180,E1 10724.427,E2 10724.427} C_VEL
LIN {X 0,Y 200.086,Z 1195.315,A -85,B 0,C 180,E1 10718.912,E2 10718.912} C_VEL
LIN {X 0,Y 200.018,Z 1196.253,A -85,B 0,C 180,E1 10714.013,E2 10714.013} C_VEL
LIN {X 0,Y 200.039,Z 1196.492,A -85,B 0,C 180,E1 10708.854,E2 10708.854} C_VEL
LIN {X 0,Y 200.027,Z 1195.884,A -85,B 0,C 180,E1 10703.398,E2 10703.398} C_VEL
LIN {X 0,Y 200.424,Z 1194.051,A -85,B 0,C 180,E1 10697.027,E2 10697.027} C_VEL
LIN {X 0,Y 201.865,Z 1191.242,A -85,B 0,C 180,E1 10690.919,E2 10690.919} C_VEL
LIN {X 0,Y 204.94,Z 1187.111,A -85,B 0,C 180,E1 10684.503,E2 10684.503} C_VEL
LIN {X 0,Y 209.462,Z 1182.172,A -85,B 0,C 180,E1 10678.647,E2 10678.647} C_VEL
LIN {X 0,Y 215.942,Z 1175.887,A -85,B 0,C 180,E1 10672.79,E2 10672.79} C_VEL
LIN {X 0,Y 225.881,Z 1167.021,A -85,B 0,C 180,E1 10666.328,E2 10666.328} C_VEL
LIN {X 0,Y 238.63,Z 1155.771,A -85,B 0,C 180,E1 10660.187,E2 10660.187} C_VEL
LIN {X 0,Y 250.267,Z 1145.545,A -85,B 0,C 180,E1 10655.805,E2 10655.805} C_VEL
LIN {X 0,Y 262.628,Z 1134.437,A -85,B 0,C 180,E1 10651.952,E2 10651.952} C_VEL
LIN {X 0,Y 278.695,Z 1119.488,A -85,B 0,C 180,E1 10647.802,E2 10647.802} C_VEL
LIN {X 0,Y 295.07,Z 1103.059,A -85,B 0,C 180,E1 10644.284,E2 10644.284} C_VEL
LIN {X 0,Y 308.152,Z 1089.209,A -85,B 0,C 180,E1 10641.878,E2 10641.878} C_VEL
LIN {X 0,Y 321.36,Z 1074.338,A -85,B 0,C 180,E1 10639.726,E2 10639.726} C_VEL
LIN {X 0,Y 335.237,Z 1057.607,A -85,B 0,C 180,E1 10637.712,E2 10637.712} C_VEL
LIN {X 0,Y 352.302,Z 1035.056,A -85,B 0,C 180,E1 10635.524,E2 10635.524} C_VEL
LIN {X 0,Y 365.272,Z 1016.086,A -85,B 0,C 180,E1 10634.03,E2 10634.03} C_VEL
LIN {X 0,Y 376.935,Z 997.475,A -85,B 0,C 180,E1 10632.812,E2 10632.812} C_VEL
LIN {X 0,Y 388.056,Z 977.971,A -85,B 0,C 180,E1 10631.735,E2 10631.735} C_VEL
LIN {X 0,Y 400.785,Z 952.92,A -85,B 0,C 180,E1 10630.603,E2 10630.603} C_VEL
LIN {X 0,Y 410.894,Z 929.883,A -85,B 0,C 180,E1 10629.765,E2 10629.765} C_VEL
LIN {X 0,Y 418.744,Z 909.557,A -85,B 0,C 180,E1 10629.158,E2 10629.158} C_VEL
LIN {X 0,Y 425.701,Z 888.879,A -85,B 0,C 180,E1 10628.646,E2 10628.646} C_VEL
LIN {X 0,Y 432.235,Z 866.043,A -85,B 0,C 180,E1 10628.189,E2 10628.189} C_VEL
LIN {X 0,Y 438.902,Z 836.168,A -85,B 0,C 180,E1 10627.708,E2 10627.708} C_VEL
LIN {X 0,Y 442.666,Z 812.681,A -85,B 0,C 180,E1 10627.365,E2 10627.365} C_VEL
LIN {X 0,Y 462.136,Z 640.41,A -85,B 0,C 180,E1 10625.058,E2 10625.058} C_VEL
LIN {X 0,Y 461.094,Z 638.27,A -85,B 0,C 180,E1 10622.859,E2 10622.859} C_VEL
LIN {X 0,Y 460.745,Z 635.8,A -85,B 0,C 180,E1 10620.373,E2 10620.373} C_VEL
LIN {X 0,Y 460.754,Z 635.932,A -85,B 0,C 180,E1 10618.881,E2 10618.881} C_VEL
LIN {X 0,Y 462.069,Z 640.323,A -85,B 0,C 180,E1 10614.54,E2 10614.54} C_VEL
LIN {X 0,Y 442.824,Z 809.947,A -85,B 0,C 180,E1 10612.281,E2 10612.281} C_VEL
LIN {X 0,Y 438.587,Z 835.698,A -85,B 0,C 180,E1 10611.906,E2 10611.906} C_VEL
LIN {X 0,Y 432.232,Z 863.3,A -85,B 0,C 180,E1 10611.403,E2 10611.403} C_VEL
LIN {X 0,Y 426.046,Z 884.934,A -85,B 0,C 180,E1 10610.904,E2 10610.904} C_VEL
LIN {X 0,Y 419.37,Z 904.843,A -85,B 0,C 180,E1 10610.353,E2 10610.353} C_VEL
LIN {X 0,Y 411.305,Z 925.756,A -85,B 0,C 180,E1 10609.662,E2 10609.662} C_VEL
LIN {X 0,Y 400.704,Z 949.813,A -85,B 0,C 180,E1 10608.705,E2 10608.705} C_VEL
LIN {X 0,Y 388.697,Z 973.134,A -85,B 0,C 180,E1 10607.561,E2 10607.561} C_VEL
LIN {X 0,Y 377.942,Z 991.883,A -85,B 0,C 180,E1 10606.466,E2 10606.466} C_VEL
LIN {X 0,Y 367.018,Z 1009.255,A -85,B 0,C 180,E1 10605.265,E2 10605.265} C_VEL
LIN {X 0,Y 355.386,Z 1026.202,A -85,B 0,C 180,E1 10603.901,E2 10603.901} C_VEL
LIN {X 0,Y 340.63,Z 1045.949,A -85,B 0,C 180,E1 10601.997,E2 10601.997} C_VEL
LIN {X 0,Y 324.244,Z 1065.647,A -85,B 0,C 180,E1 10599.624,E2 10599.624} C_VEL
LIN {X 0,Y 310.777,Z 1080.602,A -85,B 0,C 180,E1 10597.422,E2 10597.422} C_VEL
LIN {X 0,Y 297.235,Z 1094.673,A -85,B 0,C 180,E1 10594.921,E2 10594.921} C_VEL
LIN {X 0,Y 281.618,Z 1109.931,A -85,B 0,C 180,E1 10591.59,E2 10591.59} C_VEL
LIN {X 0,Y 265.525,Z 1124.484,A -85,B 0,C 180,E1 10587.511,E2 10587.511} C_VEL
LIN {X 0,Y 253.043,Z 1135.25,A -85,B 0,C 180,E1 10583.714,E2 10583.714} C_VEL
LIN {X 0,Y 241.692,Z 1144.75,A -85,B 0,C 180,E1 10579.569,E2 10579.569} C_VEL
LIN {X 0,Y 230.63,Z 1153.854,A -85,B 0,C 180,E1 10574.613,E2 10574.613} C_VEL
LIN {X 0,Y 218.593,Z 1163.782,A -85,B 0,C 180,E1 10567.47,E2 10567.47} C_VEL
LIN {X 0,Y 211.526,Z 1169.846,A -85,B 0,C 180,E1 10561.647,E2 10561.647} C_VEL
LIN {X 0,Y 206.377,Z 1174.65,A -85,B 0,C 180,E1 10555.688,E2 10555.688} C_VEL
LIN {X 0,Y 202.934,Z 1178.361,A -85,B 0,C 180,E1 10549.575,E2 10549.575} C_VEL
LIN {X 0,Y 201.013,Z 1180.981,A -85,B 0,C 180,E1 10543.52,E2 10543.52} C_VEL
LIN {X 0,Y 200.251,Z 1182.566,A -85,B 0,C 180,E1 10537.748,E2 10537.748} C_VEL
LIN {X 0,Y 200.051,Z 1183.251,A -85,B 0,C 180,E1 10532.578,E2 10532.578} C_VEL
LIN {X 0,Y 200.048,Z 1183.304,A -85,B 0,C 180,E1 10527.995,E2 10527.995} C_VEL
LIN {X 0,Y 200.224,Z 1182.661,A -85,B 0,C 180,E1 10522.54,E2 10522.54} C_VEL
LIN {X 0,Y 200.997,Z 1181.032,A -85,B 0,C 180,E1 10516.479,E2 10516.479} C_VEL
LIN {X 0,Y 202.897,Z 1178.432,A -85,B 0,C 180,E1 10510.422,E2 10510.422} C_VEL
LIN {X 0,Y 206.279,Z 1174.784,A -85,B 0,C 180,E1 10504.369,E2 10504.369} C_VEL
LIN {X 0,Y 211.171,Z 1170.201,A -85,B 0,C 180,E1 10498.612,E2 10498.612} C_VEL
LIN {X 0,Y 218.135,Z 1164.206,A -85,B 0,C 180,E1 10492.768,E2 10492.768} C_VEL
LIN {X 0,Y 228.679,Z 1155.603,A -85,B 0,C 180,E1 10486.305,E2 10486.305} C_VEL
LIN {X 0,Y 241.033,Z 1145.384,A -85,B 0,C 180,E1 10480.613,E2 10480.613} C_VEL
LIN {X 0,Y 252.318,Z 1135.957,A -85,B 0,C 180,E1 10476.446,E2 10476.446} C_VEL
LIN {X 0,Y 264.741,Z 1125.271,A -85,B 0,C 180,E1 10472.626,E2 10472.626} C_VEL
LIN {X 0,Y 280.263,Z 1111.358,A -85,B 0,C 180,E1 10468.643,E2 10468.643} C_VEL
LIN {X 0,Y 296.471,Z 1095.614,A -85,B 0,C 180,E1 10465.148,E2 10465.148} C_VEL
LIN {X 0,Y 309.868,Z 1081.761,A -85,B 0,C 180,E1 10462.655,E2 10462.655} C_VEL
LIN {X 0,Y 323.312,Z 1066.913,A -85,B 0,C 180,E1 10460.44,E2 10460.44} C_VEL
LIN {X 0,Y 337.605,Z 1049.936,A -85,B 0,C 180,E1 10458.342,E2 10458.342} C_VEL
LIN {X 0,Y 354.421,Z 1027.859,A -85,B 0,C 180,E1 10456.14,E2 10456.14} C_VEL
LIN {X 0,Y 366.732,Z 1010.018,A -85,B 0,C 180,E1 10454.689,E2 10454.689} C_VEL
LIN {X 0,Y 377.843,Z 992.411,A -85,B 0,C 180,E1 10453.466,E2 10453.466} C_VEL
LIN {X 0,Y 388.929,Z 973.119,A -85,B 0,C 180,E1 10452.339,E2 10452.339} C_VEL
LIN {X 0,Y 401.509,Z 948.52,A -85,B 0,C 180,E1 10451.141,E2 10451.141} C_VEL
LIN {X 0,Y 411.501,Z 925.834,A -85,B 0,C 180,E1 10450.244,E2 10450.244} C_VEL
LIN {X 0,Y 419.448,Z 905.273,A -85,B 0,C 180,E1 10449.564,E2 10449.564} C_VEL
LIN {X 0,Y 426.425,Z 884.474,A -85,B 0,C 180,E1 10448.988,E2 10448.988} C_VEL
LIN {X 0,Y 432.994,Z 861.343,A -85,B 0,C 180,E1 10448.461,E2 10448.461} C_VEL
LIN {X 0,Y 439.438,Z 832.265,A -85,B 0,C 180,E1 10447.947,E2 10447.947} C_VEL
LIN {X 0,Y 443.2,Z 808.932,A -85,B 0,C 180,E1 10447.611,E2 10447.611} C_VEL
LIN {X 0,Y 461.916,Z 643.899,A -85,B 0,C 180,E1 10445.413,E2 10445.413} C_VEL
LIN {X 0,Y 462.003,Z 642.217,A -85,B 0,C 180,E1 10445.247,E2 10445.247} C_VEL
LIN {X 0,Y 461.839,Z 641.477,A -85,B 0,C 180,E1 10444.874,E2 10444.874} C_VEL
LIN {X 0,Y 461.378,Z 642.18,A -85,B 0,C 180,E1 10444.264,E2 10444.264} C_VEL
LIN {X 0,Y 460.378,Z 645.446,A -85,B 0,C 180,E1 10443.028,E2 10443.028} C_VEL
LIN {X 0,Y 460.138,Z 645.723,A -85,B 0,C 180,E1 10442.447,E2 10442.447} C_VEL
LIN {X 0,Y 460.027,Z 643.783,A -85,B 0,C 180,E1 10440.374,E2 10440.374} C_VEL
LIN {X 0,Y 460.018,Z 644.241,A -85,B 0,C 180,E1 10439.377,E2 10439.377} C_VEL
LIN {X 0,Y 460.881,Z 647.723,A -85,B 0,C 180,E1 10435.84,E2 10435.84} C_VEL
LIN {X 0,Y 441.794,Z 813.563,A -85,B 0,C 180,E1 10433.66,E2 10433.66} C_VEL
LIN {X 0,Y 437.438,Z 839.769,A -85,B 0,C 180,E1 10433.284,E2 10433.284} C_VEL
LIN {X 0,Y 430.928,Z 867.495,A -85,B 0,C 180,E1 10432.846,E2 10432.846} C_VEL
LIN {X 0,Y 424.643,Z 889.096,A -85,B 0,C 180,E1 10432.427,E2 10432.427} C_VEL
LIN {X 0,Y 417.76,Z 909.302,A -85,B 0,C 180,E1 10431.945,E2 10431.945} C_VEL
LIN {X 0,Y 409.605,Z 930.14,A -85,B 0,C 180,E1 10431.345,E2 10431.345} C_VEL
LIN {X 0,Y 398.453,Z 955.103,A -85,B 0,C 180,E1 10430.46,E2 10430.46} C_VEL
LIN {X 0,Y 385.998,Z 978.943,A -85,B 0,C 180,E1 10429.402,E2 10429.402} C_VEL
LIN {X 0,Y 375.116,Z 997.695,A -85,B 0,C 180,E1 10428.394,E2 10428.394} C_VEL
LIN {X 0,Y 363.439,Z 1016.015,A -85,B 0,C 180,E1 10427.229,E2 10427.229} C_VEL
LIN {X 0,Y 350.354,Z 1034.817,A -85,B 0,C 180,E1 10425.792,E2 10425.792} C_VEL
LIN {X 0,Y 333.332,Z 1056.919,A -85,B 0,C 180,E1 10423.712,E2 10423.712} C_VEL
LIN {X 0,Y 318.987,Z 1073.866,A -85,B 0,C 180,E1 10421.732,E2 10421.732} C_VEL
LIN {X 0,Y 305.135,Z 1089.1,A -85,B 0,C 180,E1 10419.579,E2 10419.579} C_VEL
LIN {X 0,Y 290.95,Z 1103.714,A -85,B 0,C 180,E1 10417.07,E2 10417.07} C_VEL
LIN {X 0,Y 273.011,Z 1120.997,A -85,B 0,C 180,E1 10413.33,E2 10413.33} C_VEL
LIN {X 0,Y 258.348,Z 1134.179,A -85,B 0,C 180,E1 10409.661,E2 10409.661} C_VEL
LIN {X 0,Y 245.421,Z 1145.348,A -85,B 0,C 180,E1 10405.795,E2 10405.795} C_VEL
LIN {X 0,Y 233.095,Z 1155.72,A -85,B 0,C 180,E1 10401.323,E2 10401.323} C_VEL
LIN {X 0,Y 219.795,Z 1166.848,A -85,B 0,C 180,E1 10395.16,E2 10395.16} C_VEL
LIN {X 0,Y 209.452,Z 1175.535,A -85,B 0,C 180,E1 10388.708,E2 10388.708} C_VEL
LIN {X 0,Y 202.645,Z 1181.67,A -85,B 0,C 180,E1 10382.871,E2 10382.871} C_VEL
LIN {X 0,Y 197.623,Z 1186.702,A -85,B 0,C 180,E1 10376.762,E2 10376.762} C_VEL
LIN {X 0,Y 194.324,Z 1190.659,A -85,B 0,C 180,E1 10370.48,E2 10370.48} C_VEL
LIN {X 0,Y 192.645,Z 1193.44,A -85,B 0,C 180,E1 10364.426,E2 10364.426} C_VEL
LIN {X 0,Y 192.079,Z 1195.195,A -85,B 0,C 180,E1 10358.682,E2 10358.682} C_VEL
LIN {X 0,Y 192.025,Z 1196.04,A -85,B 0,C 180,E1 10353.582,E2 10353.582} C_VEL
LIN {X 0,Y 192.042,Z 1196.206,A -85,B 0,C 180,E1 10348.508,E2 10348.508} C_VEL
LIN {X 0,Y 192.039,Z 1195.547,A -85,B 0,C 180,E1 10342.822,E2 10342.822} C_VEL
LIN {X 0,Y 192.497,Z 1193.783,A -85,B 0,C 180,E1 10336.483,E2 10336.483} C_VEL
LIN {X 0,Y 194.098,Z 1190.971,A -85,B 0,C 180,E1 10330.124,E2 10330.124} C_VEL
LIN {X 0,Y 197.427,Z 1186.888,A -85,B 0,C 180,E1 10323.534,E2 10323.534} C_VEL
LIN {X 0,Y 202.364,Z 1181.896,A -85,B 0,C 180,E1 10317.415,E2 10317.415} C_VEL
LIN {X 0,Y 209.083,Z 1175.8,A -85,B 0,C 180,E1 10311.562,E2 10311.562} C_VEL
LIN {X 0,Y 218.476,Z 1167.837,A -85,B 0,C 180,E1 10305.557,E2 10305.557} C_VEL
LIN {X 0,Y 232.58,Z 1156.077,A -85,B 0,C 180,E1 10298.879,E2 10298.879} C_VEL
LIN {X 0,Y 244.798,Z 1145.792,A -85,B 0,C 180,E1 10294.407,E2 10294.407} C_VEL
LIN {X 0,Y 257.445,Z 1134.865,A -85,B 0,C 180,E1 10290.584,E2 10290.584} C_VEL
LIN {X 0,Y 270.845,Z 1122.824,A -85,B 0,C 180,E1 10287.167,E2 10287.167} C_VEL
LIN {X 0,Y 287.881,Z 1106.697,A -85,B 0,C 180,E1 10283.521,E2 10283.521} C_VEL
LIN {X 0,Y 304.323,Z 1089.789,A -85,B 0,C 180,E1 10280.55,E2 10280.55} C_VEL
LIN {X 0,Y 317.86,Z 1074.942,A -85,B 0,C 180,E1 10278.426,E2 10278.426} C_VEL
LIN {X 0,Y 331.186,Z 1059.272,A -85,B 0,C 180,E1 10276.557,E2 10276.557} C_VEL
LIN {X 0,Y 347.119,Z 1039.034,A -85,B 0,C 180,E1 10274.573,E2 10274.573} C_VEL
LIN {X 0,Y 362.535,Z 1017.06,A -85,B 0,C 180,E1 10272.855,E2 10272.855} C_VEL
LIN {X 0,Y 374.652,Z 998.095,A -85,B 0,C 180,E1 10271.64,E2 10271.64} C_VEL
LIN {X 0,Y 385.833,Z 978.841,A -85,B 0,C 180,E1 10270.603,E2 10270.603} C_VEL
LIN {X 0,Y 398.442,Z 954.665,A -85,B 0,C 180,E1 10269.53,E2 10269.53} C_VEL
LIN {X 0,Y 409.128,Z 930.746,A -85,B 0,C 180,E1 10268.681,E2 10268.681} C_VEL
LIN {X 0,Y 417.093,Z 910.49,A -85,B 0,C 180,E1 10268.092,E2 10268.092} C_VEL
LIN {X 0,Y 424.018,Z 890.314,A -85,B 0,C 180,E1 10267.605,E2 10267.605} C_VEL
LIN {X 0,Y 430.222,Z 869.211,A -85,B 0,C 180,E1 10267.19,E2 10267.19} C_VEL
LIN {X 0,Y 436.126,Z 844.825,A -85,B 0,C 180,E1 10266.796,E2 10266.796} C_VEL
LIN {X 0,Y 441.263,Z 815.679,A -85,B 0,C 180,E1 10266.373,E2 10266.373} C_VEL
LIN {X 0,Y 449.286,Z 747.097,A -85,B 0,C 180,E1 10265.462,E2 10265.462} C_VEL
LIN {X 0,Y 460.656,Z 647.333,A -85,B 0,C 180,E1 10264.142,E2 10264.142} C_VEL
LIN {X 0,Y 459.76,Z 643.741,A -85,B 0,C 180,E1 10260.249,E2 10260.249} C_VEL
LIN {X 0,Y 459.769,Z 643.954,A -85,B 0,C 180,E1 10258.878,E2 10258.878} C_VEL
LIN {X 0,Y 460.582,Z 647.491,A -85,B 0,C 180,E1 10255.442,E2 10255.442} C_VEL
LIN {X 0,Y 441.805,Z 810.338,A -85,B 0,C 180,E1 10253.308,E2 10253.308} C_VEL
LIN {X 0,Y 437.415,Z 836.625,A -85,B 0,C 180,E1 10252.935,E2 10252.935} C_VEL
LIN {X 0,Y 431.048,Z 863.791,A -85,B 0,C 180,E1 10252.452,E2 10252.452} C_VEL
LIN {X 0,Y 424.85,Z 885.207,A -85,B 0,C 180,E1 10251.974,E2 10251.974} C_VEL
LIN {X 0,Y 418.096,Z 905.115,A -85,B 0,C 180,E1 10251.441,E2 10251.441} C_VEL
LIN {X 0,Y 410.223,Z 925.323,A -85,B 0,C 180,E1 10250.795,E2 10250.795} C_VEL
LIN {X 0,Y 400.107,Z 948.101,A -85,B 0,C 180,E1 10249.925,E2 10249.925} C_VEL
LIN {X 0,Y 387.366,Z 972.807,A -85,B 0,C 180,E1 10248.767,E2 10248.767} C_VEL
LIN {X 0,Y 376.122,Z 992.154,A -85,B 0,C 180,E1 10247.67,E2 10247.67} C_VEL
LIN {X 0,Y 365.028,Z 1009.527,A -85,B 0,C 180,E1 10246.504,E2 10246.504} C_VEL
LIN {X 0,Y 352.769,Z 1027.077,A -85,B 0,C 180,E1 10245.127,E2 10245.127} C_VEL
LIN {X 0,Y 336.941,Z 1047.793,A -85,B 0,C 180,E1 10243.157,E2 10243.157} C_VEL
LIN {X 0,Y 320.714,Z 1066.755,A -85,B 0,C 180,E1 10240.891,E2 10240.891} C_VEL
LIN {X 0,Y 306.9,Z 1081.709,A -85,B 0,C 180,E1 10238.712,E2 10238.712} C_VEL
LIN {X 0,Y 292.857,Z 1095.897,A -85,B 0,C 180,E1 10236.204,E2 10236.204} C_VEL
LIN {X 0,Y 275.777,Z 1112.006,A -85,B 0,C 180,E1 10232.657,E2 10232.657} C_VEL
LIN {X 0,Y 260.47,Z 1125.321,A -85,B 0,C 180,E1 10228.873,E2 10228.873} C_VEL
LIN {X 0,Y 247.574,Z 1136.029,A -85,B 0,C 180,E1 10225.069,E2 10225.069} C_VEL
LIN {X 0,Y 235.8,Z 1145.473,A -85,B 0,C 180,E1 10220.893,E2 10220.893} C_VEL
LIN {X 0,Y 222.838,Z 1155.705,A -85,B 0,C 180,E1 10215.148,E2 10215.148} C_VEL
LIN {X 0,Y 211.668,Z 1164.349,A -85,B 0,C 180,E1 10208.574,E2 10208.574} C_VEL
LIN {X 0,Y 204.218,Z 1170.364,A -85,B 0,C 180,E1 10202.586,E2 10202.586} C_VEL
LIN {X 0,Y 198.785,Z 1175.104,A -85,B 0,C 180,E1 10196.447,E2 10196.447} C_VEL
LIN {X 0,Y 195.11,Z 1178.782,A -85,B 0,C 180,E1 10190.081,E2 10190.081} C_VEL
LIN {X 0,Y 192.944,Z 1181.571,A -85,B 0,C 180,E1 10183.18,E2 10183.18} C_VEL
LIN {X 0,Y 192.167,Z 1183.218,A -85,B 0,C 180,E1 10176.273,E2 10176.273} C_VEL
LIN {X 0,Y 192.051,Z 1183.709,A -85,B 0,C 180,E1 10170,E2 10170} C_VEL
LIN {X 0,Y 192.168,Z 1183.226,A -85,B 0,C 180,E1 10163.625,E2 10163.625} C_VEL
LIN {X 0,Y 192.927,Z 1181.621,A -85,B 0,C 180,E1 10156.819,E2 10156.819} C_VEL
LIN {X 0,Y 195.072,Z 1178.853,A -85,B 0,C 180,E1 10149.915,E2 10149.915} C_VEL
LIN {X 0,Y 198.68,Z 1175.239,A -85,B 0,C 180,E1 10143.614,E2 10143.614} C_VEL
LIN {X 0,Y 203.852,Z 1170.717,A -85,B 0,C 180,E1 10137.682,E2 10137.682} C_VEL
LIN {X 0,Y 210.817,Z 1165.064,A -85,B 0,C 180,E1 10131.935,E2 10131.935} C_VEL
LIN {X 0,Y 220.381,Z 1157.612,A -85,B 0,C 180,E1 10126.04,E2 10126.04} C_VEL
LIN {X 0,Y 234.573,Z 1146.552,A -85,B 0,C 180,E1 10119.511,E2 10119.511} C_VEL
LIN {X 0,Y 246.832,Z 1136.733,A -85,B 0,C 180,E1 10115.09,E2 10115.09} C_VEL
LIN {X 0,Y 259.669,Z 1126.104,A -85,B 0,C 180,E1 10111.261,E2 10111.261} C_VEL
LIN {X 0,Y 273.491,Z 1114.121,A -85,B 0,C 180,E1 10107.782,E2 10107.782} C_VEL
LIN {X 0,Y 291.965,Z 1096.952,A -85,B 0,C 180,E1 10103.885,E2 10103.885} C_VEL
LIN {X 0,Y 305.98,Z 1082.863,A -85,B 0,C 180,E1 10101.362,E2 10101.362} C_VEL
LIN {X 0,Y 319.796,Z 1067.989,A -85,B 0,C 180,E1 10099.166,E2 10099.166} C_VEL
LIN {X 0,Y 333.419,Z 1052.204,A -85,B 0,C 180,E1 10097.232,E2 10097.232} C_VEL
LIN {X 0,Y 349.642,Z 1031.734,A -85,B 0,C 180,E1 10095.174,E2 10095.174} C_VEL
LIN {X 0,Y 364.043,Z 1011.337,A -85,B 0,C 180,E1 10093.524,E2 10093.524} C_VEL
LIN {X 0,Y 375.576,Z 993.414,A -85,B 0,C 180,E1 10092.306,E2 10092.306} C_VEL
LIN {X 0,Y 386.37,Z 974.991,A -85,B 0,C 180,E1 10091.251,E2 10091.251} C_VEL
LIN {X 0,Y 397.277,Z 954.318,A -85,B 0,C 180,E1 10090.245,E2 10090.245} C_VEL
LIN {X 0,Y 409.221,Z 928.339,A -85,B 0,C 180,E1 10089.214,E2 10089.214} C_VEL
LIN {X 0,Y 417.556,Z 907.263,A -85,B 0,C 180,E1 10088.527,E2 10088.527} C_VEL
LIN {X 0,Y 424.69,Z 886.473,A -85,B 0,C 180,E1 10087.962,E2 10087.962} C_VEL
LIN {X 0,Y 430.897,Z 865.236,A -85,B 0,C 180,E1 10087.482,E2 10087.482} C_VEL
LIN {X 0,Y 436.701,Z 841.128,A -85,B 0,C 180,E1 10087.043,E2 10087.043} C_VEL
LIN {X 0,Y 441.793,Z 812.259,A -85,B 0,C 180,E1 10086.624,E2 10086.624} C_VEL
LIN {X 0,Y 449.978,Z 742.439,A -85,B 0,C 180,E1 10085.701,E2 10085.701} C_VEL
LIN {X 0,Y 460.835,Z 647.467,A -85,B 0,C 180,E1 10084.449,E2 10084.449} C_VEL
LIN {X 0,Y 460.138,Z 645.723,A -85,B 0,C 180,E1 10082.447,E2 10082.447} C_VEL
LIN {X 0,Y 459.887,Z 645.934,A -85,B 0,C 180,E1 10081.548,E2 10081.548} C_VEL
LIN {X 0,Y 459.431,Z 648.629,A -85,B 0,C 180,E1 10080.265,E2 10080.265} C_VEL
LIN {X 0,Y 459.092,Z 653.052,A -85,B 0,C 180,E1 10078.499,E2 10078.499} C_VEL
LIN {X 0,Y 459.135,Z 653.62,A -85,B 0,C 180,E1 10078.079,E2 10078.079} C_VEL
LIN {X 0,Y 459.489,Z 654.992,A -85,B 0,C 180,E1 10076.744,E2 10076.744} C_VEL
LIN {X 0,Y 440.978,Z 813.32,A -85,B 0,C 180,E1 10074.7,E2 10074.7} C_VEL
LIN {X 0,Y 436.57,Z 839.521,A -85,B 0,C 180,E1 10074.334,E2 10074.334} C_VEL
LIN {X 0,Y 429.987,Z 867.285,A -85,B 0,C 180,E1 10073.911,E2 10073.911} C_VEL
LIN {X 0,Y 423.654,Z 888.84,A -85,B 0,C 180,E1 10073.51,E2 10073.51} C_VEL
LIN {X 0,Y 416.514,Z 909.557,A -85,B 0,C 180,E1 10073.034,E2 10073.034} C_VEL
LIN {X 0,Y 407.843,Z 931.372,A -85,B 0,C 180,E1 10072.426,E2 10072.426} C_VEL
LIN {X 0,Y 395.309,Z 958.47,A -85,B 0,C 180,E1 10071.476,E2 10071.476} C_VEL
LIN {X 0,Y 384.104,Z 979.513,A -85,B 0,C 180,E1 10070.561,E2 10070.561} C_VEL
LIN {X 0,Y 373.091,Z 998.171,A -85,B 0,C 180,E1 10069.587,E2 10069.587} C_VEL
LIN {X 0,Y 361.254,Z 1016.423,A -85,B 0,C 180,E1 10068.458,E2 10068.458} C_VEL
LIN {X 0,Y 346.029,Z 1037.851,A -85,B 0,C 180,E1 10066.847,E2 10066.847} C_VEL
LIN {X 0,Y 329.792,Z 1058.188,A -85,B 0,C 180,E1 10064.933,E2 10064.933} C_VEL
LIN {X 0,Y 316.504,Z 1073.552,A -85,B 0,C 180,E1 10063.175,E2 10063.175} C_VEL
LIN {X 0,Y 302.502,Z 1088.627,A -85,B 0,C 180,E1 10061.099,E2 10061.099} C_VEL
LIN {X 0,Y 287.693,Z 1103.526,A -85,B 0,C 180,E1 10058.596,E2 10058.596} C_VEL
LIN {X 0,Y 269.327,Z 1120.721,A -85,B 0,C 180,E1 10054.935,E2 10054.935} C_VEL
LIN {X 0,Y 254.179,Z 1133.903,A -85,B 0,C 180,E1 10051.307,E2 10051.307} C_VEL
LIN {X 0,Y 240.763,Z 1145.072,A -85,B 0,C 180,E1 10047.462,E2 10047.462} C_VEL
LIN {X 0,Y 227.911,Z 1155.444,A -85,B 0,C 180,E1 10042.982,E2 10042.982} C_VEL
LIN {X 0,Y 213.979,Z 1166.526,A -85,B 0,C 180,E1 10036.797,E2 10036.797} C_VEL
LIN {X 0,Y 202.955,Z 1175.26,A -85,B 0,C 180,E1 10030.193,E2 10030.193} C_VEL
LIN {X 0,Y 195.515,Z 1181.527,A -85,B 0,C 180,E1 10024.055,E2 10024.055} C_VEL
LIN {X 0,Y 190.021,Z 1186.646,A -85,B 0,C 180,E1 10017.583,E2 10017.583} C_VEL
LIN {X 0,Y 186.37,Z 1190.724,A -85,B 0,C 180,E1 10010.737,E2 10010.737} C_VEL
LIN {X 0,Y 184.437,Z 1193.893,A -85,B 0,C 180,E1 10003.161,E2 10003.161} C_VEL
LIN {X 0,Y 184.026,Z 1195.583,A -85,B 0,C 180,E1 9996.109,E2 9996.109} C_VEL
LIN {X 0,Y 184.045,Z 1196.04,A -85,B 0,C 180,E1 9990.311,E2 9990.311} C_VEL
LIN {X 0,Y 184.023,Z 1195.647,A -85,B 0,C 180,E1 9984.7,E2 9984.7} C_VEL
LIN {X 0,Y 184.29,Z 1194.259,A -85,B 0,C 180,E1 9978.102,E2 9978.102} C_VEL
LIN {X 0,Y 186.048,Z 1191.166,A -85,B 0,C 180,E1 9970.139,E2 9970.139} C_VEL
LIN {X 0,Y 189.812,Z 1186.83,A -85,B 0,C 180,E1 9962.724,E2 9962.724} C_VEL
LIN {X 0,Y 195.065,Z 1181.885,A -85,B 0,C 180,E1 9956.387,E2 9956.387} C_VEL
LIN {X 0,Y 202.177,Z 1175.837,A -85,B 0,C 180,E1 9950.36,E2 9950.36} C_VEL
LIN {X 0,Y 211.583,Z 1168.288,A -85,B 0,C 180,E1 9944.474,E2 9944.474} C_VEL
LIN {X 0,Y 225.068,Z 1157.695,A -85,B 0,C 180,E1 9938.136,E2 9938.136} C_VEL
LIN {X 0,Y 239.479,Z 1146.04,A -85,B 0,C 180,E1 9932.944,E2 9932.944} C_VEL
LIN {X 0,Y 252.405,Z 1135.298,A -85,B 0,C 180,E1 9929.161,E2 9929.161} C_VEL
LIN {X 0,Y 266.359,Z 1123.192,A -85,B 0,C 180,E1 9925.722,E2 9925.722} C_VEL
LIN {X 0,Y 283.579,Z 1107.45,A -85,B 0,C 180,E1 9922.165,E2 9922.165} C_VEL
LIN {X 0,Y 300.663,Z 1090.368,A -85,B 0,C 180,E1 9919.188,E2 9919.188} C_VEL
LIN {X 0,Y 314.805,Z 1075.235,A -85,B 0,C 180,E1 9917.058,E2 9917.058} C_VEL
LIN {X 0,Y 327.938,Z 1060.15,A -85,B 0,C 180,E1 9915.291,E2 9915.291} C_VEL
LIN {X 0,Y 341.58,Z 1043.248,A -85,B 0,C 180,E1 9913.636,E2 9913.636} C_VEL
LIN {X 0,Y 358.036,Z 1020.9,A -85,B 0,C 180,E1 9911.858,E2 9911.858} C_VEL
LIN {X 0,Y 371.576,Z 1000.258,A -85,B 0,C 180,E1 9910.544,E2 9910.544} C_VEL
LIN {X 0,Y 382.744,Z 981.509,A -85,B 0,C 180,E1 9909.545,E2 9909.545} C_VEL
LIN {X 0,Y 392.962,Z 962.574,A -85,B 0,C 180,E1 9908.698,E2 9908.698} C_VEL
LIN {X 0,Y 402.8,Z 942.263,A -85,B 0,C 180,E1 9907.936,E2 9907.936} C_VEL
LIN {X 0,Y 413.661,Z 916.669,A -85,B 0,C 180,E1 9907.154,E2 9907.154} C_VEL
LIN {X 0,Y 422.453,Z 891.821,A -85,B 0,C 180,E1 9906.558,E2 9906.558} C_VEL
LIN {X 0,Y 428.818,Z 870.642,A -85,B 0,C 180,E1 9906.152,E2 9906.152} C_VEL
LIN {X 0,Y 434.333,Z 848.542,A -85,B 0,C 180,E1 9905.803,E2 9905.803} C_VEL
LIN {X 0,Y 439.674,Z 821.021,A -85,B 0,C 180,E1 9905.407,E2 9905.407} C_VEL
LIN {X 0,Y 445.227,Z 776.154,A -85,B 0,C 180,E1 9904.818,E2 9904.818} C_VEL
LIN {X 0,Y 459.268,Z 654.577,A -85,B 0,C 180,E1 9903.245,E2 9903.245} C_VEL
LIN {X 0,Y 458.786,Z 651.681,A -85,B 0,C 180,E1 9900.25,E2 9900.25} C_VEL
LIN {X 0,Y 458.788,Z 651.834,A -85,B 0,C 180,E1 9899.001,E2 9899.001} C_VEL
LIN {X 0,Y 459.209,Z 654.663,A -85,B 0,C 180,E1 9896.349,E2 9896.349} C_VEL
LIN {X 0,Y 440.944,Z 810.622,A -85,B 0,C 180,E1 9894.341,E2 9894.341} C_VEL
LIN {X 0,Y 436.472,Z 837.066,A -85,B 0,C 180,E1 9893.976,E2 9893.976} C_VEL
LIN {X 0,Y 430.038,Z 864.173,A -85,B 0,C 180,E1 9893.509,E2 9893.509} C_VEL
LIN {X 0,Y 423.803,Z 885.48,A -85,B 0,C 180,E1 9893.049,E2 9893.049} C_VEL
LIN {X 0,Y 416.763,Z 905.962,A -85,B 0,C 180,E1 9892.518,E2 9892.518} C_VEL
LIN {X 0,Y 408.432,Z 926.99,A -85,B 0,C 180,E1 9891.864,E2 9891.864} C_VEL
LIN {X 0,Y 396.925,Z 952.181,A -85,B 0,C 180,E1 9890.913,E2 9890.913} C_VEL
LIN {X 0,Y 384.95,Z 974.687,A -85,B 0,C 180,E1 9889.866,E2 9889.866} C_VEL
LIN {X 0,Y 374.015,Z 993.154,A -85,B 0,C 180,E1 9888.843,E2 9888.843} C_VEL
LIN {X 0,Y 362.762,Z 1010.461,A -85,B 0,C 180,E1 9887.71,E2 9887.71} C_VEL
LIN {X 0,Y 349.876,Z 1028.553,A -85,B 0,C 180,E1 9886.32,E2 9886.32} C_VEL
LIN {X 0,Y 332.468,Z 1050.603,A -85,B 0,C 180,E1 9884.23,E2 9884.23} C_VEL
LIN {X 0,Y 317.553,Z 1067.636,A -85,B 0,C 180,E1 9882.216,E2 9882.216} C_VEL
LIN {X 0,Y 303.997,Z 1081.983,A -85,B 0,C 180,E1 9880.163,E2 9880.163} C_VEL
LIN {X 0,Y 289.613,Z 1096.171,A -85,B 0,C 180,E1 9877.704,E2 9877.704} C_VEL
LIN {X 0,Y 272.059,Z 1112.281,A -85,B 0,C 180,E1 9874.212,E2 9874.212} C_VEL
LIN {X 0,Y 256.261,Z 1125.596,A -85,B 0,C 180,E1 9870.468,E2 9870.468} C_VEL
LIN {X 0,Y 242.893,Z 1136.305,A -85,B 0,C 180,E1 9866.682,E2 9866.682} C_VEL
LIN {X 0,Y 230.622,Z 1145.749,A -85,B 0,C 180,E1 9862.504,E2 9862.504} C_VEL
LIN {X 0,Y 217.546,Z 1155.586,A -85,B 0,C 180,E1 9856.951,E2 9856.951} C_VEL
LIN {X 0,Y 205.231,Z 1164.623,A -85,B 0,C 180,E1 9850.022,E2 9850.022} C_VEL
LIN {X 0,Y 197.287,Z 1170.637,A -85,B 0,C 180,E1 9843.882,E2 9843.882} C_VEL
LIN {X 0,Y 191.541,Z 1175.285,A -85,B 0,C 180,E1 9837.683,E2 9837.683} C_VEL
LIN {X 0,Y 187.492,Z 1178.999,A -85,B 0,C 180,E1 9831.048,E2 9831.048} C_VEL
LIN {X 0,Y 185.119,Z 1181.73,A -85,B 0,C 180,E1 9824.067,E2 9824.067} C_VEL
LIN {X 0,Y 184.204,Z 1183.417,A -85,B 0,C 180,E1 9816.858,E2 9816.858} C_VEL
LIN {X 0,Y 184.049,Z 1183.929,A -85,B 0,C 180,E1 9810.623,E2 9810.623} C_VEL
LIN {X 0,Y 184.134,Z 1183.602,A -85,B 0,C 180,E1 9804.391,E2 9804.391} C_VEL
LIN {X 0,Y 184.86,Z 1182.211,A -85,B 0,C 180,E1 9797.188,E2 9797.188} C_VEL
LIN {X 0,Y 187.263,Z 1179.273,A -85,B 0,C 180,E1 9789.366,E2 9789.366} C_VEL
LIN {X 0,Y 191.258,Z 1175.571,A -85,B 0,C 180,E1 9782.61,E2 9782.61} C_VEL
LIN {X 0,Y 196.897,Z 1170.987,A -85,B 0,C 180,E1 9776.391,E2 9776.391} C_VEL
LIN {X 0,Y 204.331,Z 1165.336,A -85,B 0,C 180,E1 9770.496,E2 9770.496} C_VEL
LIN {X 0,Y 213.971,Z 1158.227,A -85,B 0,C 180,E1 9764.743,E2 9764.743} C_VEL
LIN {X 0,Y 228.204,Z 1147.719,A -85,B 0,C 180,E1 9758.347,E2 9758.347} C_VEL
LIN {X 0,Y 242.127,Z 1137.005,A -85,B 0,C 180,E1 9753.472,E2 9753.472} C_VEL
LIN {X 0,Y 254.751,Z 1126.938,A -85,B 0,C 180,E1 9749.844,E2 9749.844} C_VEL
LIN {X 0,Y 268.243,Z 1115.638,A -85,B 0,C 180,E1 9746.545,E2 9746.545} C_VEL
LIN {X 0,Y 284.814,Z 1100.932,A -85,B 0,C 180,E1 9743.108,E2 9743.108} C_VEL
LIN {X 0,Y 302.253,Z 1083.965,A -85,B 0,C 180,E1 9740.037,E2 9740.037} C_VEL
LIN {X 0,Y 316.614,Z 1068.877,A -85,B 0,C 180,E1 9737.839,E2 9737.839} C_VEL
LIN {X 0,Y 330.06,Z 1053.656,A -85,B 0,C 180,E1 9736.002,E2 9736.002} C_VEL
LIN {X 0,Y 343.734,Z 1036.899,A -85,B 0,C 180,E1 9734.315,E2 9734.315} C_VEL
LIN {X 0,Y 360.433,Z 1014.246,A -85,B 0,C 180,E1 9732.456,E2 9732.456} C_VEL
LIN {X 0,Y 373.019,Z 995.134,A -85,B 0,C 180,E1 9731.175,E2 9731.175} C_VEL
LIN {X 0,Y 383.952,Z 976.862,A -85,B 0,C 180,E1 9730.149,E2 9730.149} C_VEL
LIN {X 0,Y 394.066,Z 958.155,A -85,B 0,C 180,E1 9729.249,E2 9729.249} C_VEL
LIN {X 0,Y 404.358,Z 936.878,A -85,B 0,C 180,E1 9728.389,E2 9728.389} C_VEL
LIN {X 0,Y 415.5,Z 910.075,A -85,B 0,C 180,E1 9727.505,E2 9727.505} C_VEL
LIN {X 0,Y 423.173,Z 888.222,A -85,B 0,C 180,E1 9726.921,E2 9726.921} C_VEL
LIN {X 0,Y 429.502,Z 867.034,A -85,B 0,C 180,E1 9726.452,E2 9726.452} C_VEL
LIN {X 0,Y 434.899,Z 845.276,A -85,B 0,C 180,E1 9726.06,E2 9726.06} C_VEL
LIN {X 0,Y 440.194,Z 817.958,A -85,B 0,C 180,E1 9725.662,E2 9725.662} C_VEL
LIN {X 0,Y 445.747,Z 773.173,A -85,B 0,C 180,E1 9725.077,E2 9725.077} C_VEL
LIN {X 0,Y 459.47,Z 654.687,A -85,B 0,C 180,E1 9723.556,E2 9723.556} C_VEL
LIN {X 0,Y 459.049,Z 651.731,A -85,B 0,C 180,E1 9720.25,E2 9720.25} C_VEL
LIN {X 0,Y 459.04,Z 652.641,A -85,B 0,C 180,E1 9719.002,E2 9719.002} C_VEL
LIN {X 0,Y 459.135,Z 653.62,A -85,B 0,C 180,E1 9718.079,E2 9718.079} C_VEL
LIN {X 0,Y 459.078,Z 654.819,A -85,B 0,C 180,E1 9717.795,E2 9717.795} C_VEL
LIN {X 0,Y 458.806,Z 657.69,A -85,B 0,C 180,E1 9717.565,E2 9717.565} C_VEL
LIN {X 0,Y 458.239,Z 662.692,A -85,B 0,C 180,E1 9717.439,E2 9717.439} C_VEL
LIN {X 0,Y 456.472,Z 676.968,A -85,B 0,C 180,E1 9717.469,E2 9717.469} C_VEL
LIN {X 0,Y 440.277,Z 813.292,A -85,B 0,C 180,E1 9715.741,E2 9715.741} C_VEL
LIN {X 0,Y 435.628,Z 840.466,A -85,B 0,C 180,E1 9715.371,E2 9715.371} C_VEL
LIN {X 0,Y 429.029,Z 867.673,A -85,B 0,C 180,E1 9714.97,E2 9714.97} C_VEL
LIN {X 0,Y 422.817,Z 888.584,A -85,B 0,C 180,E1 9714.597,E2 9714.597} C_VEL
LIN {X 0,Y 415.61,Z 909.299,A -85,B 0,C 180,E1 9714.142,E2 9714.142} C_VEL
LIN {X 0,Y 406.874,Z 931.062,A -85,B 0,C 180,E1 9713.561,E2 9713.561} C_VEL
LIN {X 0,Y 394.656,Z 957.302,A -85,B 0,C 180,E1 9712.684,E2 9712.684} C_VEL
LIN {X 0,Y 383.443,Z 978.21,A -85,B 0,C 180,E1 9711.817,E2 9711.817} C_VEL
LIN {X 0,Y 372.244,Z 997.027,A -85,B 0,C 180,E1 9710.881,E2 9710.881} C_VEL
LIN {X 0,Y 360.11,Z 1015.55,A -85,B 0,C 180,E1 9709.782,E2 9709.782} C_VEL
LIN {X 0,Y 346.945,Z 1033.897,A -85,B 0,C 180,E1 9708.476,E2 9708.476} C_VEL
LIN {X 0,Y 329.052,Z 1056.38,A -85,B 0,C 180,E1 9706.495,E2 9706.495} C_VEL
LIN {X 0,Y 314.186,Z 1073.281,A -85,B 0,C 180,E1 9704.635,E2 9704.635} C_VEL
LIN {X 0,Y 299.696,Z 1088.554,A -85,B 0,C 180,E1 9702.585,E2 9702.585} C_VEL
LIN {X 0,Y 284.824,Z 1103.167,A -85,B 0,C 180,E1 9700.186,E2 9700.186} C_VEL
LIN {X 0,Y 265.861,Z 1120.446,A -85,B 0,C 180,E1 9696.584,E2 9696.584} C_VEL
LIN {X 0,Y 250.228,Z 1133.627,A -85,B 0,C 180,E1 9693.006,E2 9693.006} C_VEL
LIN {X 0,Y 236.316,Z 1144.796,A -85,B 0,C 180,E1 9689.193,E2 9689.193} C_VEL
LIN {X 0,Y 222.92,Z 1155.168,A -85,B 0,C 180,E1 9684.718,E2 9684.718} C_VEL
LIN {X 0,Y 208.287,Z 1166.25,A -85,B 0,C 180,E1 9678.492,E2 9678.492} C_VEL
LIN {X 0,Y 196.604,Z 1174.985,A -85,B 0,C 180,E1 9671.776,E2 9671.776} C_VEL
LIN {X 0,Y 188.792,Z 1181.121,A -85,B 0,C 180,E1 9665.631,E2 9665.631} C_VEL
LIN {X 0,Y 182.781,Z 1186.284,A -85,B 0,C 180,E1 9658.923,E2 9658.923} C_VEL
LIN {X 0,Y 178.828,Z 1190.287,A -85,B 0,C 180,E1 9652,E2 9652} C_VEL
LIN {X 0,Y 176.622,Z 1193.385,A -85,B 0,C 180,E1 9644.423,E2 9644.423} C_VEL
LIN {X 0,Y 176.043,Z 1195.173,A -85,B 0,C 180,E1 9637.178,E2 9637.178} C_VEL
LIN {X 0,Y 176.051,Z 1195.731,A -85,B 0,C 180,E1 9630.976,E2 9630.976} C_VEL
LIN {X 0,Y 176.026,Z 1195.435,A -85,B 0,C 180,E1 9625.112,E2 9625.112} C_VEL
LIN {X 0,Y 176.222,Z 1194.288,A -85,B 0,C 180,E1 9618.877,E2 9618.877} C_VEL
LIN {X 0,Y 177.741,Z 1191.677,A -85,B 0,C 180,E1 9610.957,E2 9610.957} C_VEL
LIN {X 0,Y 182.019,Z 1186.988,A -85,B 0,C 180,E1 9602.166,E2 9602.166} C_VEL
LIN {X 0,Y 188.147,Z 1181.609,A -85,B 0,C 180,E1 9594.975,E2 9594.975} C_VEL
LIN {X 0,Y 195.773,Z 1175.56,A -85,B 0,C 180,E1 9588.789,E2 9588.789} C_VEL
LIN {X 0,Y 205.754,Z 1168.009,A -85,B 0,C 180,E1 9582.796,E2 9582.796} C_VEL
LIN {X 0,Y 220.515,Z 1156.971,A -85,B 0,C 180,E1 9576.188,E2 9576.188} C_VEL
LIN {X 0,Y 234.981,Z 1145.76,A -85,B 0,C 180,E1 9571.211,E2 9571.211} C_VEL
LIN {X 0,Y 248.787,Z 1134.694,A -85,B 0,C 180,E1 9567.354,E2 9567.354} C_VEL
LIN {X 0,Y 263.562,Z 1122.265,A -85,B 0,C 180,E1 9563.899,E2 9563.899} C_VEL
LIN {X 0,Y 281.704,Z 1106.022,A -85,B 0,C 180,E1 9560.356,E2 9560.356} C_VEL
LIN {X 0,Y 298.968,Z 1089.109,A -85,B 0,C 180,E1 9557.518,E2 9557.518} C_VEL
LIN {X 0,Y 313.314,Z 1074.019,A -85,B 0,C 180,E1 9555.475,E2 9555.475} C_VEL
LIN {X 0,Y 327.276,Z 1058.207,A -85,B 0,C 180,E1 9553.708,E2 9553.708} C_VEL
LIN {X 0,Y 343.907,Z 1037.739,A -85,B 0,C 180,E1 9551.837,E2 9551.837} C_VEL
LIN {X 0,Y 359.273,Z 1016.443,A -85,B 0,C 180,E1 9550.287,E2 9550.287} C_VEL
LIN {X 0,Y 371.683,Z 997.546,A -85,B 0,C 180,E1 9549.157,E2 9549.157} C_VEL
LIN {X 0,Y 382.877,Z 978.784,A -85,B 0,C 180,E1 9548.218,E2 9548.218} C_VEL
LIN {X 0,Y 395.548,Z 955.145,A -85,B 0,C 180,E1 9547.242,E2 9547.242} C_VEL
LIN {X 0,Y 406.994,Z 930.199,A -85,B 0,C 180,E1 9546.42,E2 9546.42} C_VEL
LIN {X 0,Y 415.123,Z 909.943,A -85,B 0,C 180,E1 9545.879,E2 9545.879} C_VEL
LIN {X 0,Y 422.545,Z 888.65,A -85,B 0,C 180,E1 9545.409,E2 9545.409} C_VEL
LIN {X 0,Y 429.051,Z 866.683,A -85,B 0,C 180,E1 9545.018,E2 9545.018} C_VEL
LIN {X 0,Y 435.767,Z 838.325,A -85,B 0,C 180,E1 9544.603,E2 9544.603} C_VEL
LIN {X 0,Y 440.074,Z 812.884,A -85,B 0,C 180,E1 9544.257,E2 9544.257} C_VEL
LIN {X 0,Y 457.998,Z 661.745,A -85,B 0,C 180,E1 9542.33,E2 9542.33} C_VEL
LIN {X 0,Y 457.803,Z 659.622,A -85,B 0,C 180,E1 9540.125,E2 9540.125} C_VEL
LIN {X 0,Y 457.803,Z 659.853,A -85,B 0,C 180,E1 9538.999,E2 9538.999} C_VEL
LIN {X 0,Y 457.96,Z 661.768,A -85,B 0,C 180,E1 9537.262,E2 9537.262} C_VEL
LIN {X 0,Y 440.227,Z 810.907,A -85,B 0,C 180,E1 9535.378,E2 9535.378} C_VEL
LIN {X 0,Y 435.705,Z 837.346,A -85,B 0,C 180,E1 9535.023,E2 9535.023} C_VEL
LIN {X 0,Y 429.206,Z 864.447,A -85,B 0,C 180,E1 9534.573,E2 9534.573} C_VEL
LIN {X 0,Y 422.907,Z 885.753,A -85,B 0,C 180,E1 9534.129,E2 9534.129} C_VEL
LIN {X 0,Y 415.792,Z 906.235,A -85,B 0,C 180,E1 9533.617,E2 9533.617} C_VEL
LIN {X 0,Y 407.482,Z 926.99,A -85,B 0,C 180,E1 9532.996,E2 9532.996} C_VEL
LIN {X 0,Y 396.198,Z 951.559,A -85,B 0,C 180,E1 9532.106,E2 9532.106} C_VEL
LIN {X 0,Y 384.069,Z 974.154,A -85,B 0,C 180,E1 9531.1,E2 9531.1} C_VEL
LIN {X 0,Y 372.527,Z 993.426,A -85,B 0,C 180,E1 9530.07,E2 9530.07} C_VEL
LIN {X 0,Y 361.253,Z 1010.528,A -85,B 0,C 180,E1 9528.99,E2 9528.99} C_VEL
LIN {X 0,Y 348.478,Z 1028.224,A -85,B 0,C 180,E1 9527.678,E2 9527.678} C_VEL
LIN {X 0,Y 331.581,Z 1049.443,A -85,B 0,C 180,E1 9525.754,E2 9525.754} C_VEL
LIN {X 0,Y 315.625,Z 1067.382,A -85,B 0,C 180,E1 9523.711,E2 9523.711} C_VEL
LIN {X 0,Y 301.294,Z 1082.257,A -85,B 0,C 180,E1 9521.641,E2 9521.641} C_VEL
LIN {X 0,Y 286.573,Z 1096.446,A -85,B 0,C 180,E1 9519.237,E2 9519.237} C_VEL
LIN {X 0,Y 268.548,Z 1112.556,A -85,B 0,C 180,E1 9515.809,E2 9515.809} C_VEL
LIN {X 0,Y 252.249,Z 1125.879,A -85,B 0,C 180,E1 9512.112,E2 9512.112} C_VEL
LIN {X 0,Y 238.414,Z 1136.58,A -85,B 0,C 180,E1 9508.357,E2 9508.357} C_VEL
LIN {X 0,Y 225.635,Z 1146.024,A -85,B 0,C 180,E1 9504.187,E2 9504.187} C_VEL
LIN {X 0,Y 211.416,Z 1156.254,A -85,B 0,C 180,E1 9498.351,E2 9498.351} C_VEL
LIN {X 0,Y 198.743,Z 1165.026,A -85,B 0,C 180,E1 9491.441,E2 9491.441} C_VEL
LIN {X 0,Y 190.466,Z 1170.909,A -85,B 0,C 180,E1 9485.271,E2 9485.271} C_VEL
LIN {X 0,Y 184.277,Z 1175.557,A -85,B 0,C 180,E1 9478.875,E2 9478.875} C_VEL
LIN {X 0,Y 179.968,Z 1179.169,A -85,B 0,C 180,E1 9472.197,E2 9472.197} C_VEL
LIN {X 0,Y 177.414,Z 1181.782,A -85,B 0,C 180,E1 9465.36,E2 9465.36} C_VEL
LIN {X 0,Y 176.344,Z 1183.36,A -85,B 0,C 180,E1 9458.806,E2 9458.806} C_VEL
LIN {X 0,Y 176.073,Z 1184.018,A -85,B 0,C 180,E1 9453.255,E2 9453.255} C_VEL
LIN {X 0,Y 176.059,Z 1184.113,A -85,B 0,C 180,E1 9448.047,E2 9448.047} C_VEL
LIN {X 0,Y 176.285,Z 1183.517,A -85,B 0,C 180,E1 9441.848,E2 9441.848} C_VEL
LIN {X 0,Y 177.315,Z 1181.938,A -85,B 0,C 180,E1 9434.966,E2 9434.966} C_VEL
LIN {X 0,Y 179.927,Z 1179.237,A -85,B 0,C 180,E1 9427.798,E2 9427.798} C_VEL
LIN {X 0,Y 184.22,Z 1175.643,A -85,B 0,C 180,E1 9421.115,E2 9421.115} C_VEL
LIN {X 0,Y 190.388,Z 1171.014,A -85,B 0,C 180,E1 9414.712,E2 9414.712} C_VEL
LIN {X 0,Y 198.836,Z 1165.022,A -85,B 0,C 180,E1 9408.412,E2 9408.412} C_VEL
LIN {X 0,Y 211.835,Z 1156.025,A -85,B 0,C 180,E1 9401.369,E2 9401.369} C_VEL
LIN {X 0,Y 225.516,Z 1146.202,A -85,B 0,C 180,E1 9395.772,E2 9395.772} C_VEL
LIN {X 0,Y 238.292,Z 1136.774,A -85,B 0,C 180,E1 9391.595,E2 9391.595} C_VEL
LIN {X 0,Y 252.137,Z 1126.086,A -85,B 0,C 180,E1 9387.833,E2 9387.833} C_VEL
LIN {X 0,Y 269.196,Z 1112.171,A -85,B 0,C 180,E1 9383.978,E2 9383.978} C_VEL
LIN {X 0,Y 286.458,Z 1096.733,A -85,B 0,C 180,E1 9380.702,E2 9380.702} C_VEL
LIN {X 0,Y 301.183,Z 1082.567,A -85,B 0,C 180,E1 9378.296,E2 9378.296} C_VEL
LIN {X 0,Y 315.885,Z 1067.326,A -85,B 0,C 180,E1 9376.174,E2 9376.174} C_VEL
LIN {X 0,Y 332.862,Z 1048.232,A -85,B 0,C 180,E1 9374.015,E2 9374.015} C_VEL
LIN {X 0,Y 349.282,Z 1027.45,A -85,B 0,C 180,E1 9372.156,E2 9372.156} C_VEL
LIN {X 0,Y 361.935,Z 1009.881,A -85,B 0,C 180,E1 9370.864,E2 9370.864} C_VEL
LIN {X 0,Y 373.368,Z 992.482,A -85,B 0,C 180,E1 9369.776,E2 9369.776} C_VEL
LIN {X 0,Y 385.39,Z 972.293,A -85,B 0,C 180,E1 9368.711,E2 9368.711} C_VEL
LIN {X 0,Y 398.764,Z 946.678,A -85,B 0,C 180,E1 9367.607,E2 9367.607} C_VEL
LIN {X 0,Y 408.342,Z 925.538,A -85,B 0,C 180,E1 9366.862,E2 9366.862} C_VEL
LIN {X 0,Y 416.423,Z 905.22,A -85,B 0,C 180,E1 9366.261,E2 9366.261} C_VEL
LIN {X 0,Y 423.568,Z 884.501,A -85,B 0,C 180,E1 9365.748,E2 9365.748} C_VEL
LIN {X 0,Y 430.874,Z 859.356,A -85,B 0,C 180,E1 9365.238,E2 9365.238} C_VEL
LIN {X 0,Y 436.944,Z 832.033,A -85,B 0,C 180,E1 9364.81,E2 9364.81} C_VEL
LIN {X 0,Y 440.721,Z 809.228,A -85,B 0,C 180,E1 9364.507,E2 9364.507} C_VEL
LIN {X 0,Y 458.215,Z 661.847,A -85,B 0,C 180,E1 9362.627,E2 9362.627} C_VEL
LIN {X 0,Y 458.075,Z 659.672,A -85,B 0,C 180,E1 9360.25,E2 9360.25} C_VEL
LIN {X 0,Y 458.069,Z 660.929,A -85,B 0,C 180,E1 9358.749,E2 9358.749} C_VEL
LIN {X 0,Y 458.212,Z 662.262,A -85,B 0,C 180,E1 9357.653,E2 9357.653} C_VEL
LIN {X 0,Y 456.472,Z 676.968,A -85,B 0,C 180,E1 9357.469,E2 9357.469} C_VEL
LIN {X 0,Y 455.514,Z 684.672,A -85,B 0,C 180,E1 9357.498,E2 9357.498} C_VEL
LIN {X 0,Y 452.797,Z 705.316,A -85,B 0,C 180,E1 9358.032,E2 9358.032} C_VEL
LIN {X 0,Y 451.98,Z 711.924,A -85,B 0,C 180,E1 9358.046,E2 9358.046} C_VEL
LIN {X 0,Y 439.677,Z 813.586,A -85,B 0,C 180,E1 9356.78,E2 9356.78} C_VEL
LIN {X 0,Y 434.82,Z 841.3,A -85,B 0,C 180,E1 9356.413,E2 9356.413} C_VEL
LIN {X 0,Y 428.286,Z 867.816,A -85,B 0,C 180,E1 9356.037,E2 9356.037} C_VEL
LIN {X 0,Y 421.89,Z 889.072,A -85,B 0,C 180,E1 9355.674,E2 9355.674} C_VEL
LIN {X 0,Y 414.862,Z 909.041,A -85,B 0,C 180,E1 9355.254,E2 9355.254} C_VEL
LIN {X 0,Y 406.173,Z 930.498,A -85,B 0,C 180,E1 9354.707,E2 9354.707} C_VEL
LIN {X 0,Y 393.749,Z 956.949,A -85,B 0,C 180,E1 9353.864,E2 9353.864} C_VEL
LIN {X 0,Y 382.275,Z 978.101,A -85,B 0,C 180,E1 9353.023,E2 9353.023} C_VEL
LIN {X 0,Y 370.897,Z 996.974,A -85,B 0,C 180,E1 9352.122,E2 9352.122} C_VEL
LIN {X 0,Y 359.005,Z 1014.902,A -85,B 0,C 180,E1 9351.1,E2 9351.1} C_VEL
LIN {X 0,Y 345.798,Z 1033.076,A -85,B 0,C 180,E1 9349.863,E2 9349.863} C_VEL
LIN {X 0,Y 327.659,Z 1055.597,A -85,B 0,C 180,E1 9347.962,E2 9347.962} C_VEL
LIN {X 0,Y 312.077,Z 1073.01,A -85,B 0,C 180,E1 9346.113,E2 9346.113} C_VEL
LIN {X 0,Y 297.297,Z 1088.282,A -85,B 0,C 180,E1 9344.125,E2 9344.125} C_VEL
LIN {X 0,Y 282.089,Z 1102.894,A -85,B 0,C 180,E1 9341.79,E2 9341.79} C_VEL
LIN {X 0,Y 262.624,Z 1120.172,A -85,B 0,C 180,E1 9338.272,E2 9338.272} C_VEL
LIN {X 0,Y 246.507,Z 1133.351,A -85,B 0,C 180,E1 9334.757,E2 9334.757} C_VEL
LIN {X 0,Y 232.096,Z 1144.52,A -85,B 0,C 180,E1 9330.987,E2 9330.987} C_VEL
LIN {X 0,Y 218.139,Z 1154.892,A -85,B 0,C 180,E1 9326.534,E2 9326.534} C_VEL
LIN {X 0,Y 202.791,Z 1165.974,A -85,B 0,C 180,E1 9320.278,E2 9320.278} C_VEL
LIN {X 0,Y 190.411,Z 1174.709,A -85,B 0,C 180,E1 9313.463,E2 9313.463} C_VEL
LIN {X 0,Y 182.043,Z 1180.847,A -85,B 0,C 180,E1 9307.169,E2 9307.169} C_VEL
LIN {X 0,Y 175.686,Z 1185.884,A -85,B 0,C 180,E1 9300.432,E2 9300.432} C_VEL
LIN {X 0,Y 171.352,Z 1189.848,A -85,B 0,C 180,E1 9293.377,E2 9293.377} C_VEL
LIN {X 0,Y 168.945,Z 1192.757,A -85,B 0,C 180,E1 9286.15,E2 9286.15} C_VEL
LIN {X 0,Y 168.092,Z 1194.619,A -85,B 0,C 180,E1 9278.897,E2 9278.897} C_VEL
LIN {X 0,Y 168.04,Z 1195.325,A -85,B 0,C 180,E1 9273.07,E2 9273.07} C_VEL
LIN {X 0,Y 168.049,Z 1195.394,A -85,B 0,C 180,E1 9267.954,E2 9267.954} C_VEL
LIN {X 0,Y 168.072,Z 1194.753,A -85,B 0,C 180,E1 9261.792,E2 9261.792} C_VEL
LIN {X 0,Y 168.868,Z 1192.858,A -85,B 0,C 180,E1 9254.195,E2 9254.195} C_VEL
LIN {X 0,Y 171.199,Z 1189.989,A -85,B 0,C 180,E1 9246.965,E2 9246.965} C_VEL
LIN {X 0,Y 175.433,Z 1186.066,A -85,B 0,C 180,E1 9239.898,E2 9239.898} C_VEL
LIN {X 0,Y 181.693,Z 1181.069,A -85,B 0,C 180,E1 9233.142,E2 9233.142} C_VEL
LIN {X 0,Y 189.964,Z 1174.969,A -85,B 0,C 180,E1 9226.824,E2 9226.824} C_VEL
LIN {X 0,Y 201.7,Z 1166.637,A -85,B 0,C 180,E1 9220.235,E2 9220.235} C_VEL
LIN {X 0,Y 217.503,Z 1155.28,A -85,B 0,C 180,E1 9213.69,E2 9213.69} C_VEL
LIN {X 0,Y 231.396,Z 1144.954,A -85,B 0,C 180,E1 9209.21,E2 9209.21} C_VEL
LIN {X 0,Y 245.015,Z 1134.415,A -85,B 0,C 180,E1 9205.597,E2 9205.597} C_VEL
LIN {X 0,Y 260.256,Z 1121.986,A -85,B 0,C 180,E1 9202.199,E2 9202.199} C_VEL
LIN {X 0,Y 278.767,Z 1105.861,A -85,B 0,C 180,E1 9198.757,E2 9198.757} C_VEL
LIN {X 0,Y 296.43,Z 1088.955,A -85,B 0,C 180,E1 9195.992,E2 9195.992} C_VEL
LIN {X 0,Y 311.189,Z 1073.741,A -85,B 0,C 180,E1 9193.992,E2 9193.992} C_VEL
LIN {X 0,Y 325.404,Z 1057.931,A -85,B 0,C 180,E1 9192.284,E2 9192.284} C_VEL
LIN {X 0,Y 342.174,Z 1037.634,A -85,B 0,C 180,E1 9190.494,E2 9190.494} C_VEL
LIN {X 0,Y 357.706,Z 1016.441,A -85,B 0,C 180,E1 9189.006,E2 9189.006} C_VEL
LIN {X 0,Y 370.312,Z 997.513,A -85,B 0,C 180,E1 9187.915,E2 9187.915} C_VEL
LIN {X 0,Y 381.793,Z 978.51,A -85,B 0,C 180,E1 9187.003,E2 9187.003} C_VEL
LIN {X 0,Y 394.172,Z 955.686,A -85,B 0,C 180,E1 9186.097,E2 9186.097} C_VEL
LIN {X 0,Y 405.685,Z 931.062,A -85,B 0,C 180,E1 9185.314,E2 9185.314} C_VEL
LIN {X 0,Y 414.372,Z 909.669,A -85,B 0,C 180,E1 9184.765,E2 9184.765} C_VEL
LIN {X 0,Y 421.593,Z 889.193,A -85,B 0,C 180,E1 9184.332,E2 9184.332} C_VEL
LIN {X 0,Y 428.056,Z 867.713,A -85,B 0,C 180,E1 9183.965,E2 9183.965} C_VEL
LIN {X 0,Y 434.692,Z 840.704,A -85,B 0,C 180,E1 9183.581,E2 9183.581} C_VEL
LIN {X 0,Y 439.457,Z 813.257,A -85,B 0,C 180,E1 9183.218,E2 9183.218} C_VEL
LIN {X 0,Y 454.392,Z 689.418,A -85,B 0,C 180,E1 9181.677,E2 9181.677} C_VEL
LIN {X 0,Y 456.855,Z 668.834,A -85,B 0,C 180,E1 9181.414,E2 9181.414} C_VEL
LIN {X 0,Y 456.823,Z 667.56,A -85,B 0,C 180,E1 9180,E2 9180} C_VEL
LIN {X 0,Y 456.819,Z 667.869,A -85,B 0,C 180,E1 9178.997,E2 9178.997} C_VEL
LIN {X 0,Y 456.824,Z 668.906,A -85,B 0,C 180,E1 9178.18,E2 9178.18} C_VEL
LIN {X 0,Y 439.639,Z 811.298,A -85,B 0,C 180,E1 9176.417,E2 9176.417} C_VEL
LIN {X 0,Y 434.942,Z 838.38,A -85,B 0,C 180,E1 9176.063,E2 9176.063} C_VEL
LIN {X 0,Y 428.431,Z 865.045,A -85,B 0,C 180,E1 9175.634,E2 9175.634} C_VEL
LIN {X 0,Y 422.161,Z 886.026,A -85,B 0,C 180,E1 9175.214,E2 9175.214} C_VEL
LIN {X 0,Y 414.975,Z 906.507,A -85,B 0,C 180,E1 9174.721,E2 9174.721} C_VEL
LIN {X 0,Y 406.578,Z 927.262,A -85,B 0,C 180,E1 9174.123,E2 9174.123} C_VEL
LIN {X 0,Y 395.168,Z 951.83,A -85,B 0,C 180,E1 9173.267,E2 9173.267} C_VEL
LIN {X 0,Y 382.428,Z 975.231,A -85,B 0,C 180,E1 9172.261,E2 9172.261} C_VEL
LIN {X 0,Y 371.211,Z 993.698,A -85,B 0,C 180,E1 9171.306,E2 9171.306} C_VEL
LIN {X 0,Y 359.393,Z 1011.361,A -85,B 0,C 180,E1 9170.229,E2 9170.229} C_VEL
LIN {X 0,Y 345.462,Z 1030.302,A -85,B 0,C 180,E1 9168.858,E2 9168.858} C_VEL
LIN {X 0,Y 327.49,Z 1052.15,A -85,B 0,C 180,E1 9166.889,E2 9166.889} C_VEL
LIN {X 0,Y 312.543,Z 1068.569,A -85,B 0,C 180,E1 9165.045,E2 9165.045} C_VEL
LIN {X 0,Y 297.981,Z 1083.329,A -85,B 0,C 180,E1 9163.026,E2 9163.026} C_VEL
LIN {X 0,Y 281.279,Z 1098.995,A -85,B 0,C 180,E1 9160.388,E2 9160.388} C_VEL
LIN {X 0,Y 262.12,Z 1115.323,A -85,B 0,C 180,E1 9156.823,E2 9156.823} C_VEL
LIN {X 0,Y 246.996,Z 1127.27,A -85,B 0,C 180,E1 9153.46,E2 9153.46} C_VEL
LIN {X 0,Y 232.768,Z 1137.862,A -85,B 0,C 180,E1 9149.7,E2 9149.7} C_VEL
LIN {X 0,Y 216.497,Z 1149.427,A -85,B 0,C 180,E1 9144.373,E2 9144.373} C_VEL
LIN {X 0,Y 201.621,Z 1159.314,A -85,B 0,C 180,E1 9138.061,E2 9138.061} C_VEL
LIN {X 0,Y 191.433,Z 1166.05,A -85,B 0,C 180,E1 9132.359,E2 9132.359} C_VEL
LIN {X 0,Y 182.803,Z 1171.834,A -85,B 0,C 180,E1 9125.95,E2 9125.95} C_VEL
LIN {X 0,Y 175.805,Z 1176.817,A -85,B 0,C 180,E1 9118.538,E2 9118.538} C_VEL
LIN {X 0,Y 170.586,Z 1181.086,A -85,B 0,C 180,E1 9109.162,E2 9109.162} C_VEL
LIN {X 0,Y 168.675,Z 1183.181,A -85,B 0,C 180,E1 9101.627,E2 9101.627} C_VEL
LIN {X 0,Y 168.126,Z 1184.178,A -85,B 0,C 180,E1 9095.118,E2 9095.118} C_VEL
LIN {X 0,Y 168.06,Z 1184.441,A -85,B 0,C 180,E1 9088.977,E2 9088.977} C_VEL
LIN {X 0,Y 168.268,Z 1183.91,A -85,B 0,C 180,E1 9082.145,E2 9082.145} C_VEL
LIN {X 0,Y 169.479,Z 1182.204,A -85,B 0,C 180,E1 9074.254,E2 9074.254} C_VEL
LIN {X 0,Y 172.36,Z 1179.506,A -85,B 0,C 180,E1 9066.767,E2 9066.767} C_VEL
LIN {X 0,Y 177.094,Z 1175.869,A -85,B 0,C 180,E1 9059.752,E2 9059.752} C_VEL
LIN {X 0,Y 183.814,Z 1171.19,A -85,B 0,C 180,E1 9053.096,E2 9053.096} C_VEL
LIN {X 0,Y 193.262,Z 1164.925,A -85,B 0,C 180,E1 9046.413,E2 9046.413} C_VEL
LIN {X 0,Y 208.083,Z 1155.116,A -85,B 0,C 180,E1 9038.884,E2 9038.884} C_VEL
LIN {X 0,Y 221.38,Z 1146.027,A -85,B 0,C 180,E1 9033.796,E2 9033.796} C_VEL
LIN {X 0,Y 235.074,Z 1136.293,A -85,B 0,C 180,E1 9029.565,E2 9029.565} C_VEL
LIN {X 0,Y 251.302,Z 1124.14,A -85,B 0,C 180,E1 9025.45,E2 9025.45} C_VEL
LIN {X 0,Y 270.393,Z 1108.592,A -85,B 0,C 180,E1 9021.475,E2 9021.475} C_VEL
LIN {X 0,Y 285.282,Z 1095.486,A -85,B 0,C 180,E1 9018.863,E2 9018.863} C_VEL
LIN {X 0,Y 299.544,Z 1082.002,A -85,B 0,C 180,E1 9016.668,E2 9016.668} C_VEL
LIN {X 0,Y 314.19,Z 1067.07,A -85,B 0,C 180,E1 9014.664,E2 9014.664} C_VEL
LIN {X 0,Y 331.927,Z 1047.349,A -85,B 0,C 180,E1 9012.527,E2 9012.527} C_VEL
LIN {X 0,Y 347.65,Z 1027.715,A -85,B 0,C 180,E1 9010.837,E2 9010.837} C_VEL
LIN {X 0,Y 360.025,Z 1010.806,A -85,B 0,C 180,E1 9009.633,E2 9009.633} C_VEL
LIN {X 0,Y 371.607,Z 993.473,A -85,B 0,C 180,E1 9008.582,E2 9008.582} C_VEL
LIN {X 0,Y 383.304,Z 974.164,A -85,B 0,C 180,E1 9007.591,E2 9007.591} C_VEL
LIN {X 0,Y 396.531,Z 949.556,A -85,B 0,C 180,E1 9006.55,E2 9006.55} C_VEL
LIN {X 0,Y 407.31,Z 926.142,A -85,B 0,C 180,E1 9005.747,E2 9005.747} C_VEL
LIN {X 0,Y 415.623,Z 905.476,A -85,B 0,C 180,E1 9005.158,E2 9005.158} C_VEL
LIN {X 0,Y 422.84,Z 884.755,A -85,B 0,C 180,E1 9004.665,E2 9004.665} C_VEL
LIN {X 0,Y 430.183,Z 859.727,A -85,B 0,C 180,E1 9004.176,E2 9004.176} C_VEL
LIN {X 0,Y 436.346,Z 832.28,A -85,B 0,C 180,E1 9003.762,E2 9003.762} C_VEL
LIN {X 0,Y 440.164,Z 809.469,A -85,B 0,C 180,E1 9003.468,E2 9003.468} C_VEL
LIN {X 0,Y 457.085,Z 669.029,A -85,B 0,C 180,E1 9001.724,E2 9001.724} C_VEL
LIN {X 0,Y 457.099,Z 667.619,A -85,B 0,C 180,E1 9000.125,E2 9000.125} C_VEL
LIN {X 0,Y 457.076,Z 669.327,A -85,B 0,C 180,E1 8998.571,E2 8998.571} C_VEL
LIN {X 0,Y 451.98,Z 711.924,A -85,B 0,C 180,E1 8998.046,E2 8998.046} C_VEL
LIN {X 0,Y 451.025,Z 719.628,A -85,B 0,C 180,E1 8998.078,E2 8998.078} C_VEL
LIN {X 0,Y 448.35,Z 740.27,A -85,B 0,C 180,E1 8998.625,E2 8998.625} C_VEL
LIN {X 0,Y 447.534,Z 746.879,A -85,B 0,C 180,E1 8998.641,E2 8998.641} C_VEL
LIN {X 0,Y 439.124,Z 814.574,A -85,B 0,C 180,E1 8997.814,E2 8997.814} C_VEL
LIN {X 0,Y 433.715,Z 843.925,A -85,B 0,C 180,E1 8997.435,E2 8997.435} C_VEL
LIN {X 0,Y 427.607,Z 868.263,A -85,B 0,C 180,E1 8997.103,E2 8997.103} C_VEL
LIN {X 0,Y 421.113,Z 889.559,A -85,B 0,C 180,E1 8996.755,E2 8996.755} C_VEL
LIN {X 0,Y 413.454,Z 910.945,A -85,B 0,C 180,E1 8996.321,E2 8996.321} C_VEL
LIN {X 0,Y 402.592,Z 936.908,A -85,B 0,C 180,E1 8995.667,E2 8995.667} C_VEL
LIN {X 0,Y 390.836,Z 960.676,A -85,B 0,C 180,E1 8994.904,E2 8994.904} C_VEL
LIN {X 0,Y 380.501,Z 979.315,A -85,B 0,C 180,E1 8994.181,E2 8994.181} C_VEL
LIN {X 0,Y 368.897,Z 998.211,A -85,B 0,C 180,E1 8993.307,E2 8993.307} C_VEL
LIN {X 0,Y 355.767,Z 1017.578,A -85,B 0,C 180,E1 8992.228,E2 8992.228} C_VEL
LIN {X 0,Y 337.987,Z 1041.006,A -85,B 0,C 180,E1 8990.603,E2 8990.603} C_VEL
LIN {X 0,Y 323.66,Z 1057.986,A -85,B 0,C 180,E1 8989.138,E2 8989.138} C_VEL
